// TwinCAT 3 PLC project EpicsComModule
// ProgramVersion: 3.1.4022.2
// libraries:
//   Tc2_EtherCAT, * (Beckhoff Automation GmbH)
//   Tc2_Standard, * (Beckhoff Automation GmbH)
//   Tc2_System, * (Beckhoff Automation GmbH)
//   Tc2_TcpIp, * (Beckhoff Automation GmbH)
//   Tc2_Utilities, * (Beckhoff Automation GmbH)
//   Tc3_Interfaces, * (Beckhoff Automation GmbH)
//   Tc3_Module, * (Beckhoff Automation GmbH)
// project tree:
//   Data types/ DUT_AxisStatus_v0_01.TcDUT, E_ConnectionSteps.TcDUT, E_ServerSteps.TcDUT, DUT_ComSettings.TcDUT
//   Global Variables/ Global_Variables.TcGVL
//   / PlcTaskCom.TcTTO
//   POUs/DUT_Support/ FB_Read_DUT_AxisStatus_v0_01.TcPOU
//   POUs/ FB_ServerApplication.TcPOU, FB_ServerConnection.TcPOU, FB_Server.TcPOU, FB_StreamBufferToADSBuffer.TcPOU, FB_ValidCommand.TcPOU, FB_ADSBufferToStreamBuffer.TcPOU, MAIN.TcPOU, README.TcPOU
//   POUs/Helper POUs/ CheckBounds.TcPOU, FB_FindChar.TcPOU, FB_FrameFifo.TcPOU, FB_LogFifo.TcPOU, F_RemoveBytesFromBuffer.TcPOU
//   POUs/Static Command support/ FB_GetStaticADR.TcPOU, FB_ParseStaticCommand.TcPOU, FB_ParseStringToSymInfo.TcPOU, FB_SetStaticADSPort.TcPOU, FB_SetStaticADR.TcPOU, FB_ParseCommandOption.TcPOU

CONFIGURATION EpicsComModule
    RESOURCE PLC ON TwinCAT3
        TASK PlcTaskCom(INTERVAL := T#1ms, PRIORITY := 26);
        PROGRAM MAIN WITH PlcTaskCom : MAIN;
    END_RESOURCE
END_CONFIGURATION

// ---- Data types/DUT_AxisStatus_v0_01.TcDUT
TYPE DUT_AxisStatus_v0_01:
STRUCT
    bEnable: BOOL;
    bReset: BOOL;
    bExecute: BOOL;
    nCommand: UINT;
    nCmdData: UINT;
    fVelocity: LREAL;
    fPosition: LREAL;
    fAcceleration: LREAL;
    fDeceleration: LREAL;
    bJogFwd: BOOL;
    bJogBwd: BOOL;
    bLimitFwd: BOOL;
    bLimitBwd: BOOL;
    fOverride: LREAL:=100;
    bHomeSensor: BOOL;
    bEnabled: BOOL;
    bError: BOOL;
    nErrorId: UDINT;
    fActVelocity: LREAL;
    fActPosition: LREAL;
    fActDiff: LREAL;
    bHomed:BOOL;
    bBusy:BOOL;
END_STRUCT
END_TYPE

// ---- Data types/E_ConnectionSteps.TcDUT
TYPE E_ConnectionSteps :
(
    eCONNECTION_STATE_IDLE,
    eCONNECTION_STATE_CONNECT_START,
    eCONNECTION_STATE_CONNECT_WAIT,
    eCONNECTION_STATE_DATAEXCHANGE,
    eCONNECTION_STATE_CLOSE_START,
    eCONNECTION_STATE_CLOSE_WAIT,
    eCONNECTION_STATE_ERROR
);
END_TYPE

// ---- Data types/E_ServerSteps.TcDUT
TYPE E_ServerSteps :
(
    eSERVER_STATE_IDLE,
    eSERVER_STATE_LISTENER_OPEN_START,
    eSERVER_STATE_LISTENER_OPEN_WAIT,
    eSERVER_STATE_REMOTE_CLIENTS_COMM,
    eSERVER_STATE_REMOTE_CLIENTS_CLOSE,
    eSERVER_STATE_LISTENER_CLOSE_START,
    eSERVER_STATE_LISTENER_CLOSE_WAIT,
    eSERVER_STATE_ERROR
);
END_TYPE

// ---- Data types/DUT_ComSettings.TcDUT
TYPE DUT_ComSettings :
STRUCT
    nConnectionIndex:UDINT:=0;
    nADSPort:INT:=851;
    bReturnData:BOOL:=FALSE;
    bReturnVarName:BOOL:=FALSE;
END_STRUCT
END_TYPE

// ---- Global Variables/Global_Variables.TcGVL
VAR_GLOBAL CONSTANT
    MAX_CLIENT_CONNECTIONS                  : UDINT(1..20) := 5;
    PLCPRJ_BUFFER_SIZE                      : UDINT := 20000;(* Max. internal fifo/receiver buffer size *)
    PLCPRJ_RECEIVE_POLLING_TIME             : TIME := T#1MS; //Changed from example where it was 1000ms. => epics timeout all the time!
    PLCPRJ_RECEIVE_TIMEOUT                  : TIME := T#0S;

    (* Some project specific error codes *)
    PLCPRJ_ERROR_RECEIVE_TIMEOUT            : UDINT := 16#8101;(* Receive timeout *)
    PLCPRJ_ERROR_SENDFIFO_OVERFLOW          : UDINT := 16#8102;(* Send fifo overflow *)
    PLCPRJ_ERROR_RECFIFO_OVERFLOW           : UDINT := 16#8103;(* Receive fifo overflow *)

    //EPICS related constants
    EPICS_MAX_FRAME_SIZE                    : INT :=1400; //Max size of variable string (for communication with epics) Arrays can be divided in several frames/stings (atleast for reading operation)
    EPICS_ARRAY_DELIMITER                   : STRING :=',';
    EPICS_COMMAND_DELIMITER                 : STRING := ';';
    EPICS_READ_CMD                          : STRING:= '?';
    EPICS_WRITE_CMD                         : STRING:= '=';
    EPICS_ACK_STRING                        : STRING:='OK';
    EPICS_ASCII_DOT                         : BYTE:=46;
    EPICS_ASCII_LN                          : BYTE:=10;
    EPICS_ASCII_CR                          : BYTE:=13;
    EPICS_ASCII_COMMA                       : BYTE:=44;     // Must be same as EPICS_ARRAY_DELIMITER. This variable should be autoamtically genrated instead. Maybe in next version?!
    EPICS_ASCII_ZERO                        : BYTE:=48;
    EPICS_ASCII_ONE                         : BYTE:=49;
    EPICS_ASCII_EQUAL                       : BYTE:=61;     // Must be same as EPICS_WRITE_CMD. This variable should be autoamtically genrated instead. Maybe in next version?!
    EPICS_ASCII_QUESTIONMARK                : BYTE:=63;     // Must be same as EPICS_READ_CMD. This variable should be autoamtically genrated instead. Maybe in next version?!
    EPICS_ASCII_COMMAND_DELIMITER           : BYTE:=59;     // Must be same as EPICS_COMMAND_DELIMITER. This variable should be autoamtically genrated instead. Maybe in next version?!
    EPICS_COM_TIMEOUT                       : TIME:=T#1S;   // Not used yet
    EPICS_MAX_STACKED_STATIC_COMMANDS       : INT:=5;       // Maximum options to command

    //Command Options
    EPICS_COMMAND_OPTION_DELIMITER          : STRING := '/';        //Used for static commands that should not excute symboliclly
    EPICS_COMMAND_OPTION_ADSPORT            : STRING := 'ADSPORT';  //USED to set ADS port from command. Applicable only for this command

    //Static Commands
    EPICS_STATIC_COMMAND_TRIGGER            : STRING := '.';        //Setting for return of data for write commands (data instead of "OK;"). Applicable only for this command
    EPICS_STATIC_COMMAND_THIS               : STRING := 'THIS.';    //Setting for return of data for write commands (data instead of "OK;"). Applicable only for this command
    EPICS_STATIC_COMMAND_THIS_PATH          : STRING := 'Main.fbServer.aApplications';  //Setting for return of data for write commands (data instead of "OK;"). Applicable only for this command
    EPICS_STATIC_COMMAND_ADR                : STRING := 'ADR.';     //Setting for return of data for write commands (data instead of "OK;"). Applicable only for this command

END_VAR

VAR_GLOBAL
        EPICS_SAMPLE_TIME                   : INT:=1;       // The EPICS COM module will be executed every EPICS_SAMPLE_TIME cycle
        EPICS_FORMAT_ASCII                  : BOOL:=TRUE;   // Not used yet. Binary transfer of data is not currently supported.
END_VAR

// ---- POUs/MAIN.TcPOU
///#########################################################
///Main POU for TCP/IP based EPICS-interface. The TCP/IP server related code is based on Beckhoff sample code. Changes and additions have been made to this code for the general purpose EPICS interface.
///
/// Library:
///
///
/// Global Variables:
/// - EPICS_MAX_FRAME_SIZE
/// - EPICS_ARRAY_DELIMITER
/// - EPICS_COMMAND_DELIMITER
/// - PLCPRJ_BUFFER_SIZE
///
/// Data types:
///
/// External functions:
///     - TC2_Standard lib
///     - Tc2_Utilities lib
///     - Tc2_System lib
///
///
///###########################################################

PROGRAM MAIN
VAR
    sVersion: STRING:='0.9.1';
END_VAR
VAR
    sSrvNetID   : T_AmsNetID    := '';(* TwinCAT TCP/IP server network address *)
    bEnable     : BOOL := TRUE;(* TRUE => Enable server data exchange, FALSE => Disable *)
    bLog        : BOOL := FALSE;(* TRUE => Enable message/error log, FALSE => Disable *)

    fbServer    : FB_Server := (    sLocalHost :=  '0.0.0.0' (*Own (server) IP address!  '192.168.40.106'*),
                                    nLocalPort := 5000,(* Own (server) port number! *)
                                    sPrefix := 'SERVER::' );

    fbCloseAll  : FB_SocketCloseAll;
    bInitialize : BOOL := TRUE;

    //Included utilities in EpicsComModule
    fbNTShutdown: NT_Shutdown;
    fbNTAbortShutdown:NT_AbortShutdown;
    iCounter:INT:=0;
    bErrorWritten:BOOL:=FALSE;
    sErrorMessage:STRING(255);
END_VAR

//Delay execution
IF EPICS_SAMPLE_TIME>100 THEN
    EPICS_SAMPLE_TIME:=100;
ELSIF  EPICS_SAMPLE_TIME<1 THEN
    EPICS_SAMPLE_TIME:=1;
END_IF

iCounter:=iCounter+1;
IF iCounter>=EPICS_SAMPLE_TIME THEN  //Possability to change communcation execution speed from EPICS (via the global variable EPICS_SAMPLE_TIME)
    iCounter:=0;
    (* On PLC reset or program download close all created/opened sockets/connections *)
    fbCloseAll( sSrvNetID := sSrvNetID, bExecute:= bInitialize );
    IF fbCloseAll.bError AND NOT bErrorWritten THEN
        sErrorMessage:=UDINT_TO_STRING(fbCloseAll.nErrId);
        ADSLOGSTR( ADSLOG_MSGTYPE_ERROR, 'EPICSComModule: fbCloseAll failed with errorId %s.', sErrorMessage);
        bErrorWritten:=TRUE;
    END_IF
    IF fbCloseAll.bBusy OR fbCloseAll.bError THEN
        RETURN;
    END_IF
    bErrorWritten:=FALSE;
    bInitialize := FALSE;
    fbServer( sSrvNetID := sSrvNetID, bEnable := bEnable, bLog := bLog );
END_IF

//Execution of utilities Action
Utilities();

ACTION Utilities:
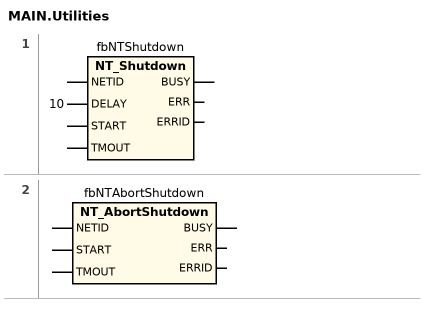
// NETWORK 1
//   fbNTShutdown: Included utilities in EpicsComModule
fbNTShutdown(DELAY := 10); // NT_Shutdown

// NETWORK 2
fbNTAbortShutdown(); // NT_AbortShutdown
END_ACTION

END_PROGRAM

// ---- POUs/FB_Server.TcPOU
///#########################################################
///FB that handles TCP/IP server and the client connections. The code is based on Beckhoff sample code. However changes and additions have been made to this code for the general purpose EPICS interface.
///
///
/// Library:
///
/// Global Variables:
/// - EPICS_MAX_FRAME_SIZE
/// - EPICS_ARRAY_DELIMITER
/// - EPICS_COMMAND_DELIMITER
/// - PLCPRJ_BUFFER_SIZE
///
/// Data types:
///
/// External functions:
///     - TC2_Standard lib
///     - Tc2_Utilities lib
///     - Tc2_System lib
///
///###########################################################

FUNCTION_BLOCK FB_Server
VAR
    sVersion: STRING:='0.9.1';
END_VAR
VAR_INPUT
    sSrvNetID       : T_AmsNetID    := '';(* TwinCAT TCP/IP server network address *)
    sLocalHost      : T_IPv4Addr    := '127.0.0.1';(* Own IP address! *)
    nLocalPort      : UDINT         := 0;(* Server port number *)
    bEnable         : BOOL          := FALSE;(* TRUE => enable server data exchange, FALSE => disable *)
    tReconnect      : TIME          := T#3S;(* Reopen new listener socket after this time *)
    bLog            : BOOL          := FALSE;(* TRUE => Enable log message output, FALSE => Disable *)
    sPrefix         : STRING        := 'SERVER::';(* Log message description string (allows the identification of log message source) *)
END_VAR
VAR_OUTPUT
    bListening      : BOOL          := FALSE;(* Listener socket state *)
    nAccepted       : UDINT         := 0;(* Max. number of accepted client connections *)
END_VAR
VAR
    aApplications   : ARRAY[1..MAX_CLIENT_CONNECTIONS] OF FB_ServerApplication;(* Server application control function blocks *)
    aConnections    : ARRAY[1..MAX_CLIENT_CONNECTIONS] OF FB_ServerConnection :=
                                                    [   (sPrefix := 'SERVER1::'),
                                                        (sPrefix := 'SERVER2::'),
                                                        (sPrefix := 'SERVER3::'),
                                                        (sPrefix := 'SERVER4::'),
                                                        (sPrefix := 'SERVER5::') ];(* Server connection/data exchange control function blocks *)
    aTx             : ARRAY[1..MAX_CLIENT_CONNECTIONS] OF FB_FrameFifo;(* TX fifo *)
    aRx             : ARRAY[1..MAX_CLIENT_CONNECTIONS] OF FB_FrameFifo;(* RX fifo *)
    aLog            : ARRAY[1..MAX_CLIENT_CONNECTIONS] OF FB_LogFifo;(* Listener log message fifo *)
    fbListen        : FB_SocketListen;
    fbClose         : FB_SocketClose;
    fbLog           : FB_LogFifo;
    fbListenTimer   : TON;
    bReset          : BOOL := FALSE;
    eStep           : E_ServerSteps;
    i               : UDINT;
END_VAR



CASE eStep OF
    eSERVER_STATE_IDLE:
        IF bEnable XOR bListening THEN
            IF bEnable THEN
                fbListenTimer( IN := TRUE );
                IF fbListenTimer.Q THEN
                    fbListenTimer( IN := FALSE, PT := tReconnect );

                    fbLog.Clear( sPrefix := sPrefix, bLog := bLog );(* Clear listener log fifo *)
                    bReset := FALSE;

                    eStep := eSERVER_STATE_LISTENER_OPEN_START;
                END_IF
            ELSE
                eStep := eSERVER_STATE_REMOTE_CLIENTS_CLOSE;
            END_IF
        ELSIF bListening THEN
            eStep := eSERVER_STATE_REMOTE_CLIENTS_COMM;
        ELSE
            fbListenTimer( IN := FALSE, PT := T#0S );
            bReset := FALSE;
        END_IF

    eSERVER_STATE_LISTENER_OPEN_START:
        fbListen(  bExecute := FALSE  );
        fbListen(   sSrvNetID := sSrvNetID,
                    sLocalHost := sLocalHost,
                    nLocalPort := nLocalPort,
                    bExecute := TRUE );
        eStep := eSERVER_STATE_LISTENER_OPEN_WAIT;

    eSERVER_STATE_LISTENER_OPEN_WAIT:
        fbListen( bExecute := FALSE );
        IF NOT fbListen.bBusy THEN
            IF NOT fbListen.bError THEN
                bListening  := TRUE;
                fbLog.Message( sMessage := 'Listener socket opened!', hSocket := fbListen.hListener );
                eStep := eSERVER_STATE_IDLE;
            ELSE
                fbLog.Error( sMessage := 'FB_SocketListen()', nErrId := fbListen.nErrId );
                eStep := eSERVER_STATE_ERROR;
            END_IF
        END_IF

    eSERVER_STATE_REMOTE_CLIENTS_COMM:
        eStep := eSERVER_STATE_IDLE;
        nAccepted := 0;

        FOR i:= 1 TO MAX_CLIENT_CONNECTIONS DO
            aApplications[i].nConnectionIndex:=i;
            aConnections[i]( fbTx := aTx[i], fbRx := aRx[i], fbLog := aLog[i],
                            hListener := fbListen.hListener, bReset := bReset,
                            sSrvNetID := sSrvNetID, bEnable := bEnable, bLog := bLog );
            IF bReset THEN
                bReset := FALSE;
                eStep := eSERVER_STATE_REMOTE_CLIENTS_CLOSE;
                EXIT;
            END_IF

            IF aConnections[i].bAccepted THEN
                aApplications[i]( fbTx := aTx[i], fbRx := aRx[i], fbLog := aLog[i]);
                nAccepted := nAccepted + 1;(* Count the number of connected remote clients *)
                aApplications[i].bReset:=FALSE;
            ELSE
                    aApplications[i].bReset:=TRUE;
                    aApplications[i]( fbTx := aTx[i], fbRx := aRx[i], fbLog := aLog[i]);
            END_IF


        END_FOR

    eSERVER_STATE_REMOTE_CLIENTS_CLOSE:
        nAccepted := 0;
        FOR i:= 1 TO MAX_CLIENT_CONNECTIONS DO
            (* Close all remote client (accepted) sockets *)
            aConnections[i]( fbTx := aTx[i], fbRx := aRx[i], fbLog := aLog[i],
                            hListener := fbListen.hListener, bReset := bReset,
                            sSrvNetID := sSrvNetID, bEnable := FALSE, bLog := bLog );
            IF aConnections[i].bAccepted THEN
                nAccepted := nAccepted + 1;(* Count the number of connected remote clients *)
            END_IF
        END_FOR

        (* Check if all remote client sockets are closed *)
        IF nAccepted = 0 THEN
            eStep := eSERVER_STATE_LISTENER_CLOSE_START; (* Close listener socket too *)
        END_IF

    eSERVER_STATE_LISTENER_CLOSE_START:
        fbLog.Message( sMessage := 'Closing listener socket!', hSocket := fbListen.hListener );
        fbClose( bExecute := FALSE );
        fbClose( sSrvNetID := sSrvNetID, hSocket := fbListen.hListener, bExecute:= TRUE );
        eStep := eSERVER_STATE_LISTENER_CLOSE_WAIT;

    eSERVER_STATE_LISTENER_CLOSE_WAIT:
        fbClose( bExecute := FALSE );
        IF NOT fbClose.bBusy THEN
            bListening := FALSE;
            nAccepted := 0;
            IF NOT fbClose.bError THEN
                eStep := eSERVER_STATE_IDLE;
            ELSE
                fbLog.Error( sMessage := 'FB_SocketClose(listener)', nErrId := fbListen.nErrID );
                eStep := eSERVER_STATE_ERROR;
            END_IF
        END_IF

    eSERVER_STATE_ERROR:
        IF bListening THEN
            eStep := eSERVER_STATE_REMOTE_CLIENTS_CLOSE;
        ELSE
            eStep := eSERVER_STATE_IDLE;
        END_IF

END_CASE

END_FUNCTION_BLOCK

// ---- POUs/FB_ServerApplication.TcPOU
///#########################################################
///FB that handles one EPICS connection of TCP/IP.
/// The main functionallity of this function block is to parse commands from EPICS or other serial device.
///
/// Library:
///
///
/// Global Variables:
/// - EPICS_MAX_FRAME_SIZE
/// - EPICS_ARRAY_DELIMITER
/// - EPICS_COMMAND_DELIMITER
/// - PLCPRJ_BUFFER_SIZE
///
/// Data types:
///
/// External functions:
///     - TC2_Standard lib
///     - Tc2_Utilities lib
///     - Tc2_System lib
///
///###########################################################
FUNCTION_BLOCK FB_ServerApplication
VAR
    sVersion: STRING:='0.9.1';
    sFeatures: STRING:='stv1';
END_VAR
VAR_IN_OUT
    fbTx        : FB_FrameFifo;(* TX fifo *)
    fbRx        : FB_FrameFifo;(* RX fifo *)
    fbLog       : FB_LogFifo;(* Log message fifo *)
END_VAR

VAR_INPUT
    nConnectionIndex:UDINT:=0;
    bReset: BOOL;
END_VAR

VAR
    //Settings
    nADSPort                            : UINT:=851;
    nState                              :INT:=0;

    bExecuteWriteBufferToEPICS:BOOL:=FALSE;
    bInStaticSection:BOOL:=FALSE;
    bReadCmd: BOOL:=FALSE;
    bWriteCmd: BOOL:=FALSE;
    bStaticGetADRCommand    :   BOOL:=FALSE;
    bStaticTHISCommand      :   BOOL:=FALSE;

    //FB:s
    fbAdsReadValue: Tc2_System.ADSREAD;
    fbAdsWriteValue: Tc2_System.ADSWRITE;
    fbParseADSBufferToStream:FB_ADSBufferToStreamBuffer;
    fbParseStreamBufferToADS:FB_StreamBufferToADSBuffer;
    fbStateTimoutTimer:TON;
    fbSymInfoByName:Tc2_Utilities.PLC_ReadSymInfoByName;
    fbValidCommand:FB_ValidCommand;
    fbParseCommandOption:FB_ParseCommandOption;
    fbParseStringToSymInfo: FB_ParseStringToSymInfo;
    stSettings: DUT_ComSettings;
    fbFincChar: FB_FindChar;
    //buffers
    byteADSBuffer       : ARRAY[0..PLCPRJ_BUFFER_SIZE] OF BYTE;
    byteCommandBuffer   : ARRAY[0..PLCPRJ_BUFFER_SIZE] OF BYTE; (* Byte buffer*)
    byteFrameBuffer     : ARRAY[0..EPICS_MAX_FRAME_SIZE] OF BYTE;

    //Strings
    sTemp: STRING;
    sAckString: STRING;
    psCommandBufferString: POINTER TO STRING; //string to point into byte buffer
    sVariableName: STRING;

    //Ints
    nBytesInCommandBuffer:DINT;
    nADSBytesToRead: DINT;
    nIndexEndOfCommand: DINT;
    nIndex1:INT:=0;
    nLength: INT;

    //Error handling
    sComBufferAtError: STRING;
    sError: STRING(255);
    sSubErrorString:STRING(255);
    bErrorMessageSent: BOOL:=FALSE;
    bErrorOld: BOOL;
    nErrorCounter: INT;
    stSymInfo:SYMINFOSTRUCT;
    nStatricCommandCounter: INT;
    sGetStaticADR:STRING(255):='';
    iEmptyCounter: INT;
    nFrameBufferIndex: INT;
    nCleanBytes: DINT;
    sVariableName_THIS: STRING(INT#255);
    sVarName: STRING(INT#255);
    nLengthSubString: INT;
END_VAR

VAR_OUTPUT
    nErrorId: UDINT;
    bError: BOOL;
END_VAR



//Typical command string: "ADSPORT=851/Main.M1.fPosition=100;ADSPORT=852/Main.iCounter?;linefeed"

psCommandBufferString :=ADR(byteCommandBuffer[0]); //Used for debugging to see byte buffer as string
stSettings.nConnectionIndex:=nConnectionIndex;

//State 1: Get new info from recieve buffer. Wait for complete command = ";"
IF nState=0 THEN //Only get new data from buffer if free mem
    fbRx.RemoveHead(bGet := ADR(byteCommandBuffer[nBytesInCommandBuffer]), nReadBufferSize:=SIZEOF(byteCommandBuffer)-nBytesInCommandBuffer);(* Fetch string from rx fifo *)
    IF fbRx.bOk THEN(* Success *)
        nBytesInCommandBuffer:=nBytesInCommandBuffer+DINT_TO_INT(fbRx.nReadCount); //Seems buffer always returns one byte less thann count?
        //fbLog.Error( sMessage := concat(str1:='State 1a: ', str2:=PSTRING_TO_STRING(psCommandBufferString)), nErrID := nBytesInCommandBuffer );
    END_IF
END_IF

IF  nBytesInCommandBuffer>0 AND NOT (nState=1) THEN
    fbValidCommand(nBytesInCommandBuffer:=nBytesInCommandBuffer,pbCommandBuffer:=ADR(byteCommandBuffer));
    //fbLog.Error( sMessage := concat(str1:='State 1b: ', str2:=PSTRING_TO_STRING(psCommandBufferString)), nErrID := nBytesInCommandBuffer );
    IF  fbValidCommand.bValid THEN
        nIndexEndOfCommand:=fbValidCommand.nIndexEndOfCommand;
        nState:=1;
    END_IF
END_IF

//State 2: Check for Command Options
IF (nState=1) THEN
    //Reset defaults
    nADSPort:=stSettings.nADSPort;
    nStatricCommandCounter:=0;
    bInStaticSection:=TRUE;
    REPEAT
        nStatricCommandCounter:=nStatricCommandCounter+1;
        nIndex1:=find(STR1:=PSTRING_TO_STRING(psCommandBufferString),STR2:=EPICS_COMMAND_OPTION_DELIMITER);

        IF nIndex1>0 AND nIndex1<=nIndexEndOfCommand THEN
            fbParseCommandOption(nCommandEndIndex:=nIndex1,byteCommandBuffer:=byteCommandBuffer,nBytesInCommandBuffer:=nBytesInCommandBuffer,nIndexEndOfCommand:=nIndexEndOfCommand);
            IF NOT fbParseCommandOption.bError THEN
                IF len(fbParseCommandOption.sStaticCommand)>0 THEN
                    //*****EPICS_COMMAND_OPTION_ADSPORT
                    IF find(STR1:=fbParseCommandOption.sStaticCommand,STR2:=EPICS_COMMAND_OPTION_ADSPORT)>0 THEN
                        IF fbParseCommandOption.bWriteCommand THEN
                            nADSPort:=STRING_TO_UINT(fbParseCommandOption.sStaticValue);
                        END_IF
                    END_IF
                END_IF
            ELSE
                bError:=fbParseCommandOption.bError;
                sSubErrorString:=fbParseCommandOption.sSubErrorString;
                nErrorId:=fbParseCommandOption.nErrorId;
            END_IF
        ELSE
            bInStaticSection:=FALSE;
        END_IF
    UNTIL nBytesInCommandBuffer<1 OR (NOT bInStaticSection) OR bError OR nStatricCommandCounter>EPICS_MAX_STACKED_STATIC_COMMANDS OR nIndex1=0
    END_REPEAT
    IF NOT bError THEN
        nState:=2;
    END_IF
    //fbLog.Error( sMessage := concat(str1:='State 2: ', str2:=PSTRING_TO_STRING(psCommandBufferString)), nErrID := nBytesInCommandBuffer );
END_IF

//State 3: Check if Static Commands
IF (nState=2) THEN
    bStaticTHISCommand:=FALSE;
    bStaticGetADRCommand:=FALSE;
    nIndex1:=find(STR1:=PSTRING_TO_STRING(psCommandBufferString),STR2:=EPICS_STATIC_COMMAND_TRIGGER);
    IF (nIndex1=1) THEN
         //Command EPICS_STATIC_COMMAND_THIS = "#THIS."
        nIndex1:=find(STR1:=PSTRING_TO_STRING(psCommandBufferString),STR2:=EPICS_STATIC_COMMAND_THIS);
        IF (nIndex1=2) THEN   //Command should be = "#THIS."
            //=
            nIndex1:=find(STR1:=PSTRING_TO_STRING(psCommandBufferString),STR2:=EPICS_WRITE_CMD);        //=
            IF nIndex1<1 OR nIndex1 > nIndexEndOfCommand THEN
                nIndex1:=find(STR1:=PSTRING_TO_STRING(psCommandBufferString),STR2:=EPICS_READ_CMD); //?
            END_IF
            //Remove static commands and build variable name to this fb. (this.stSettings.nPort=>Main.fbServer.aApplications[nConnectionIndex].stSettings.nPort)
            stemp:=left(str:=PSTRING_TO_STRING(psCommandBufferString),SIZE:=nIndex1-1);
            stemp:=right(str:=sTemp,size:=len(sTemp)-(len(EPICS_STATIC_COMMAND_TRIGGER)+len(EPICS_STATIC_COMMAND_THIS)));
            sVariableName_THIS:=concat(STR1:=EPICS_STATIC_COMMAND_THIS_PATH,STR2:='[');
            sVariableName_THIS:=concat(STR1:=sVariableName_THIS,STR2:=UDINT_TO_STRING(nConnectionIndex));
            sVariableName_THIS:=concat(STR1:=sVariableName_THIS,STR2:='].');
            sVariableName_THIS:=concat(STR1:=sVariableName_THIS,STR2:=sTemp);
            bStaticTHISCommand:=TRUE;
            //Don't clean up this command. Will be done in subsequent steps
        ELSE
             //Command EPICS_STATIC_COMMAND_THIS = "#ADR."
            nIndex1:=find(STR1:=PSTRING_TO_STRING(psCommandBufferString),STR2:=EPICS_STATIC_COMMAND_ADR);
            IF (nIndex1=2) THEN   //Command should be = "#ADR."
                //= write. Expect a command like:  "#ADR.1,1,1,1=200;"
                nIndex1:=find(STR1:=PSTRING_TO_STRING(psCommandBufferString),STR2:=EPICS_WRITE_CMD);        //=
                IF (nIndex1>0) AND ((nIndex1-1) < nIndexEndOfCommand) THEN
                    bWriteCmd:=TRUE;
                ELSE
                    //? read. Expect a command like:  "#ADR.1,1,1,1?;" => ask for value, or "#ADR.Main.M1.bEnable?;"=> ask for adress
                    nIndex1:=find(STR1:=PSTRING_TO_STRING(psCommandBufferString),STR2:=EPICS_READ_CMD);     //?
                    IF ((nIndex1>0) AND (nIndex1-1) < nIndexEndOfCommand) THEN
                        bReadCmd:=TRUE;
                    END_IF
                END_IF
                IF bReadCmd OR bWriteCmd THEN
                    sVariableName:=left(str:=PSTRING_TO_STRING(psCommandBufferString),SIZE:=nIndex1-1);
                    sVariableName:=right(str:=sVariableName,size:=len(sVariableName)-(len(EPICS_STATIC_COMMAND_TRIGGER)+len(EPICS_STATIC_COMMAND_ADR)));
                    //Check if symbol or abs adress
                    nLengthSubString:=(len(EPICS_STATIC_COMMAND_ADR)+len(EPICS_STATIC_COMMAND_TRIGGER));
                    fbFincChar(pbBuffer:=ADR(byteCommandBuffer[0]),nLength:=nIndex1,cFind:=EPICS_ASCII_DOT,nStartIndex:=nLengthSubString+2);
                    IF ((fbFincChar.nIndex>nLengthSubString) AND (fbFincChar.nIndex-1) <nIndexEndOfCommand) THEN
                        bStaticGetADRCommand:=TRUE;
                        nState:=4;  // return abs.-adress for symbolic adress
                    ELSE
                        fbParseStringToSymInfo(sAdress:=sVariableName);
                        IF NOT fbParseStringToSymInfo.bError THEN
                            stSymInfo:=fbParseStringToSymInfo.stSymInfo;
                            nState:=5;
                        ELSE
                            bError:=fbParseStringToSymInfo.bError;
                            nErrorId:=fbParseStringToSymInfo.nErrorId;
                            sSubErrorString:=fbParseStringToSymInfo.sSubErrorString;
                        END_IF
                    END_IF
                    IF NOT F_RemoveBytesFromBuffer(nIndex1,byteCommandBuffer:=byteCommandBuffer,nBytesInCommandBuffer:=nBytesInCommandBuffer,nIndexEndOfCommand:=nIndexEndOfCommand) THEN
                            bError:=TRUE;
                            nErrorId:=301;
                            sSubErrorString:='State 3: Failed to clear buffer (read).';
                    END_IF
                END_IF
            END_IF
        END_IF
    END_IF
    IF (NOT bError) AND (nState<3) THEN
        nState:=3;
    END_IF
    //fbLog.Error( sMessage := concat(str1:='State 3: ', str2:=PSTRING_TO_STRING(psCommandBufferString)), nErrID := nBytesInCommandBuffer );
END_IF

//State 4: Find symbolic variable name in cmd
IF (nState=3) THEN
    //check if read cmd
    bReadCmd:=FALSE;
    bWriteCmd:=FALSE;
    nIndex1:=find(STR1:=PSTRING_TO_STRING(psCommandBufferString),STR2:=EPICS_READ_CMD);
    IF nIndex1>0 AND nIndex1<= nIndexEndOfCommand THEN
        sVariableName:=left(STR:=PSTRING_TO_STRING(psCommandBufferString), SIZE:=nIndex1-1);
        //Clear buffer
        IF F_RemoveBytesFromBuffer(nIndex1,byteCommandBuffer:=byteCommandBuffer,nBytesInCommandBuffer:=nBytesInCommandBuffer,nIndexEndOfCommand:=nIndexEndOfCommand) THEN
            bReadCmd:=TRUE;
        ELSE
            bError:=TRUE;
            nErrorId:=402;
            sSubErrorString:='State 4: Failed to clear buffer (read).';
        END_IF
    ELSE
        nIndex1:=find(STR1:=PSTRING_TO_STRING(psCommandBufferString),STR2:=EPICS_WRITE_CMD);
        IF nIndex1>0 AND nIndex1<=nIndexEndOfCommand THEN
            sVariableName:=left(STR:=PSTRING_TO_STRING(psCommandBufferString), SIZE:=nIndex1-1);
            IF F_RemoveBytesFromBuffer(nIndex1,byteCommandBuffer:=byteCommandBuffer,nBytesInCommandBuffer:=nBytesInCommandBuffer,nIndexEndOfCommand:=nIndexEndOfCommand) THEN
                bWriteCmd:=TRUE;
            ELSE
                bError:=TRUE;
                nErrorId:=403;
                sSubErrorString:='State 4: Failed to clear buffer (write).';
            END_IF
        END_IF
    END_IF
    IF bWriteCmd OR bReadCmd THEN
        nState:=4;
    END_IF
    IF NOT bError THEN
        IF NOT (nState=4) THEN
            bError:=TRUE;
            nErrorId:=401;
            sSubErrorString:='State 4: No read or write command identified.';
        END_IF
    END_IF;
    fbSymInfoByName(START:=FALSE);
    //fbLog.Error( sMessage := concat(str1:='State 4: ', str2:=PSTRING_TO_STRING(psCommandBufferString)), nErrID := nBytesInCommandBuffer );
END_IF


//State 5: Get symbolic information over ADS
IF (nState=4) THEN
    //If static command "THIS" then use other variable name
    IF bStaticTHISCommand THEN
        sVarName:=sVariableName_THIS;
    ELSE
        sVarName:=sVariableName;
    END_IF
    fbSymInfoByName(
            PORT:= nADSPort,
            SYMNAME:= sVarName,
            START:= TRUE,
            TMOUT:=T#100MS);

        (*Wait until it's done or if an error occurs*)
        IF NOT fbSymInfoByName.ERR THEN
            IF NOT fbSymInfoByName.BUSY THEN
                nState:=5;
                stSymInfo:=fbSymInfoByName.SYMINFO;
                fbAdsReadValue(read:=FALSE);
                IF bStaticGetADRCommand THEN // jump over next state and prepare information to be sent
                    sGetStaticADR:='';
                    sGetStaticADR:=CONCAT(str1:=sGetStaticADR,str2:='16#');
                    sGetStaticADR:=CONCAT(str1:=sGetStaticADR,str2:=DWORD_TO_HEXSTR(stSymInfo.idxGroup,1,FALSE));
                    sGetStaticADR:=CONCAT(str1:=sGetStaticADR,str2:=EPICS_ARRAY_DELIMITER);
                    sGetStaticADR:=CONCAT(str1:=sGetStaticADR,str2:='16#');
                    sGetStaticADR:=CONCAT(str1:=sGetStaticADR,str2:=DWORD_TO_HEXSTR(stSymInfo.idxOffset,1,FALSE));
                    sGetStaticADR:=CONCAT(str1:=sGetStaticADR,str2:=EPICS_ARRAY_DELIMITER);
                    sGetStaticADR:=CONCAT(str1:=sGetStaticADR,str2:=DINT_TO_STRING(stSymInfo.byteSize));
                    sGetStaticADR:=CONCAT(str1:=sGetStaticADR,str2:=EPICS_ARRAY_DELIMITER);
                    sGetStaticADR:=CONCAT(str1:=sGetStaticADR,str2:=DINT_TO_STRING(stSymInfo.adsDataType));
                    nFrameBufferIndex:=len(sGetStaticADR);
                    stSymInfo.byteSize:=len(str:=sGetStaticADR);        //Fake size
                    memcpy(destAddr:=ADR(byteADSBuffer[0]),srcAddr:=ADR(sGetStaticADR),n:=stSymInfo.byteSize);  //Copy to output buffer
                    stSymInfo.adsDataType :=ADST_STRING;                //Fake string
                    bReadCmd:=TRUE;
                    nState:=8;                                          //Jump to state 9
                    bExecuteWriteBufferToEPICS:=TRUE;                   //Execute write directly size all info is prepared
                END_IF
            END_IF
        ELSE
            bError:=TRUE;
            nErrorId:=fbSymInfoByName.ERRID;
            sSubErrorString:=concat(str1:='State 5: Failed to get symbolic information for variable:',STR2:=sVariableName);
        END_IF;
        //fbLog.Error( sMessage := concat(str1:='State 5: ', str2:=PSTRING_TO_STRING(psCommandBufferString)), nErrID := nBytesInCommandBuffer );
END_IF

//State 6: Convert stream buffer to ADS buffer (WRITE)
IF (nState=5) AND bWriteCmd THEN
    //fbLog.Error( sMessage := concat(str1:='State 6: ', str2:=PSTRING_TO_STRING(psCommandBufferString)), nErrID := nBytesInCommandBuffer );
    fbParseStreamBufferToADS(bExecute:=TRUE,symbolInfo:=stSymInfo,nBufferToParseLength:=nIndexEndOfCommand,fbLog:=fbLog,byteASCIIBufferToParse:=byteCommandBuffer,byteBinayBufferOutput:=byteADSBuffer);
    IF NOT fbParseStreamBufferToADS.bError  THEN
        IF NOT fbParseStreamBufferToADS.bBusy THEN
            nCleanBytes:=fbParseStreamBufferToADS.nASCIIBytesParsed;
            IF nCleanBytes>0 AND nCleanBytes+fbParseStreamBufferToADS.nASCIIBytesParsed < PLCPRJ_BUFFER_SIZE-255 THEN
                F_RemoveBytesFromBuffer(nCleanBytes,byteCommandBuffer:=byteCommandBuffer,nBytesInCommandBuffer:=nBytesInCommandBuffer,nIndexEndOfCommand:=nIndexEndOfCommand);
                fbAdsWriteValue(WRITE:=FALSE);
                nState:=6;
                fbParseStreamBufferToADS(bExecute:=FALSE,symbolInfo:=stSymInfo,nBufferToParseLength:=nIndexEndOfCommand,fbLog:=fbLog,byteASCIIBufferToParse:=byteCommandBuffer,byteBinayBufferOutput:=byteADSBuffer);
            ELSE
                bError:=TRUE;
                nErrorID:=701;
                sSubErrorString:='State 6: Buffer index out of range.';
            END_IF
        END_IF;
    ELSE
        bError:=TRUE;
        nErrorId:=fbParseStreamBufferToADS.nErrorId;
        sSubErrorString:='State 6: Failed to parse ASCII buffer to ADS buffer.';
    END_IF;

END_IF

//State 7: Write ADS data
IF (nState=6) THEN
    IF stSymInfo.byteSize>=fbParseStreamBufferToADS.nBinaryBytesWritten THEN //Ensure right size of variable
        fbAdsWriteValue(
            PORT:= nADSPort,
            IDXGRP:= stSymInfo.idxGroup,
            IDXOFFS:= stSymInfo.idxOffset,
            LEN:= fbParseStreamBufferToADS.nBinaryBytesWritten,
            SRCADDR:=ADR(byteADSBuffer[0]) ,
            WRITE:= TRUE,
            TMOUT:= T#5S,
        );
        IF NOT fbAdsWriteValue.ERR THEN
            IF NOT fbAdsWriteValue.BUSY THEN
                fbAdsWriteValue(Write:=FALSE);
                nState:=7;
            END_IF
        ELSE
            bError:=TRUE;
            nErrorId:=fbAdsWriteValue.ERRID;
            sSubErrorString:='State 7: Failed ADS write command.';
        END_IF
    ELSE
            bError:=TRUE;
            nErrorId:=711;
            sSubErrorString:='State 7: Size missmatch between ASCII data and variable size.';
    END_IF
    //fbLog.Error( sMessage := concat(str1:='State 7: ', str2:=PSTRING_TO_STRING(psCommandBufferString)), nErrID := nBytesInCommandBuffer );
END_IF

//State 8: Read data over ADS
IF (((nState=5) AND bReadCmd) OR ((nState=7) AND bWriteCmd AND stSettings.bReturnData)) THEN
    IF(stSymInfo.byteSize>PLCPRJ_BUFFER_SIZE-255) THEN
        nADSBytesToRead:=PLCPRJ_BUFFER_SIZE-255;
    ELSE
        nADSBytesToRead:=stSymInfo.byteSize;
    END_IF
    fbAdsReadValue(
        PORT:= nADSPort,
        IDXGRP:= stSymInfo.idxGroup,
        IDXOFFS:=stSymInfo.idxOffset,
        LEN:= nADSBytesToRead,
        DESTADDR:=ADR(byteADSBuffer),
        Read:= TRUE,
        TMOUT:= T#100MS,
     );

     IF NOT fbAdsReadValue.ERR THEN
        IF NOT fbAdsReadValue.BUSY THEN
            fbAdsReadValue(READ:=FALSE);
            bExecuteWriteBufferToEPICS:=TRUE;
            nState:=8;
        END_IF
    ELSE
        bError:=TRUE;
        nErrorId:=fbAdsReadValue.ERRID;
        sSubErrorString:='State 8: Failed ADS read command.';
    END_IF;
    //fbLog.Error( sMessage := concat(str1:='State 6a: ', str2:=PSTRING_TO_STRING(psCommandBufferString)), nErrID := nBytesInCommandBuffer );
END_IF

//State 9: Parse stream and send to buffer if needed
fbParseADSBufferToStream(bExecute:=bExecuteWriteBufferToEPICS,symbolInfo:=stSymInfo,fbTx:=fbTx,fbLog:=fbLog,byteBufferToSend:=byteADSBuffer,bReturnVariableName:=stSettings.bReturnVarName, sVariableName:=sVariableName, byteFrameBuffer:=byteFrameBuffer,nFrameBufferIndex:=nFrameBufferIndex);
IF (nState=8) THEN
    bExecuteWriteBufferToEPICS:=TRUE;
    IF NOT fbParseADSBufferToStream.bError THEN
        IF NOT fbParseADSBufferToStream.bBusy THEN
            nState:=9;
            bExecuteWriteBufferToEPICS:=FALSE;
        END_IF
    ELSE
        bError:=TRUE;
        nErrorId:=fbParseADSBufferToStream.nErrorId;
        sSubErrorString:='State 9: Failed to parse ADS buffer to ASCII buffer.';
    END_IF
    //fbLog.Error( sMessage := concat(str1:='State 6b: ', str2:=PSTRING_TO_STRING(psCommandBufferString)), nErrID := nBytesInCommandBuffer );
END_IF


//State10: Send data to EPICS
IF ((nState=9) OR ((nState=7) AND NOT stSettings.bReturnData AND bWriteCmd)) THEN
    IF bWriteCmd AND NOT stSettings.bReturnData THEN
        //Copy 'OK' sting to output buffer
        nFrameBufferIndex:=len(STR:=EPICS_ACK_STRING);
        memcpy(destAddr:=ADR(byteFrameBuffer[0]),srcAddr:=ADR(EPICS_ACK_STRING), nFrameBufferIndex);
    ELSIF bReadCmd OR stSettings.bReturnData THEN
        IF nFrameBufferIndex> EPICS_MAX_FRAME_SIZE-3 THEN  //must be space for atleast 3 bytes  (';crlf')
            fbTx.AddTail( bPut := ADR(byteFrameBuffer[0]), nWriteCount:=nFrameBufferIndex );(* Put string to the tx fifo *)
            IF NOT fbTx.bOk THEN(* TX fifo overflow => log error *)
                bError:=TRUE;
                nErrorId:=801;
                sSubErrorString:='State 7c: TX buffer overflow.';
            END_IF
            nFrameBufferIndex:=0;
        END_IF
    END_IF;
    nCleanBytes:=0;
    //check for semi-colon and add it to output buffer
    IF(byteCommandBuffer[nIndexEndOfCommand]=F_ToASC(str:=EPICS_COMMAND_DELIMITER)) THEN //CR or LF
        byteFrameBuffer[nFrameBufferIndex]:=byteCommandBuffer[nIndexEndOfCommand];
        nFrameBufferIndex:=nFrameBufferIndex+1;
        nCleanBytes:=nCleanBytes+1;
        IF(byteCommandBuffer[nIndexEndOfCommand+1]=EPICS_ASCII_LN OR byteCommandBuffer[nIndexEndOfCommand+1]=EPICS_ASCII_CR) THEN //CR or LF
            byteFrameBuffer[nFrameBufferIndex]:=byteCommandBuffer[nIndexEndOfCommand+1];
            nFrameBufferIndex:=nFrameBufferIndex+1;
            nCleanBytes:=nCleanBytes+1;
        END_IF;
        IF(byteCommandBuffer[nIndexEndOfCommand+2]=EPICS_ASCII_LN OR byteCommandBuffer[nIndexEndOfCommand+2]=EPICS_ASCII_CR) THEN //CR or LF
            byteFrameBuffer[nFrameBufferIndex]:=byteCommandBuffer[nIndexEndOfCommand+2];
            nFrameBufferIndex:=nFrameBufferIndex+1;
            nCleanBytes:=nCleanBytes+1;
        END_IF;

        //Send OK or data to output queue
        fbTx.AddTail( bPut := ADR(byteFrameBuffer[0]), nWriteCount:=nFrameBufferIndex );(* Put string to the tx fifo *)
        IF NOT fbTx.bOk THEN(* TX fifo overflow => log error *)
            bError:=TRUE;
            nErrorId:=802;
            sSubErrorString:='State 8: TX buffer overflow.';
        ELSE
            nState:=10;
        END_IF
    ELSE
            bError:=TRUE;
            nErrorId:=803;
            sSubErrorString:='State 8: Semi-colon missing.';
    END_IF
    //fbLog.Error( sMessage := concat(str1:='State : ', str2:=PSTRING_TO_STRING(psCommandBufferString)), nErrID := nBytesInCommandBuffer );
END_IF


//State 11: Clean ";" and CR or LN from buffer, also see if extra zeros(=0) in buffer..
IF (nState=10) THEN
    IF nCleanBytes>0 THEN
        F_RemoveBytesFromBuffer(nCleanBytes,byteCommandBuffer:=byteCommandBuffer,nBytesInCommandBuffer:=nBytesInCommandBuffer,nIndexEndOfCommand:=nIndexEndOfCommand);
    END_IF;
    //Clean extra bytes/spaces Check if extra empty bytes
    iEmptyCounter:=0;
    IF nBytesInCommandBuffer>0 THEN
        WHILE byteCommandBuffer[iEmptyCounter]=0 AND iEmptyCounter<nBytesInCommandBuffer DO
            iEmptyCounter:=iEmptyCounter+1;
        END_WHILE
        //remove bytes
        F_RemoveBytesFromBuffer(iEmptyCounter,byteCommandBuffer:=byteCommandBuffer,nBytesInCommandBuffer:=nBytesInCommandBuffer,nIndexEndOfCommand:=nIndexEndOfCommand);
    END_IF

    nState:=11;
    //fbLog.Error( sMessage := concat(str1:='State 8: ', str2:=PSTRING_TO_STRING(psCommandBufferString)), nErrID := nBytesInCommandBuffer );
END_IF

// Command ready: Start over
IF (nState=11) THEN
    nState:=0;
    bReadCmd:=FALSE;
    bWriteCmd:=FALSE;
    nIndexEndOfCommand:=0;
    bExecuteWriteBufferToEPICS:=FALSE;
    //fbLog.Error( sMessage := concat(str1:='State 9: ', str2:=PSTRING_TO_STRING(psCommandBufferString)), nErrID := nBytesInCommandBuffer );
    IF nBytesInCommandBuffer<0 THEN
        nBytesInCommandBuffer:=0;
    END_IF
    fbAdsReadValue(read:=FALSE);
    fbAdsWriteValue(WRITE:=FALSE);
    fbSymInfoByName(start:=FALSE);

END_IF

//Ensure that communiucation not hangs du to stuck in one state

fbStateTimoutTimer(In:=(nState>0 OR nBytesInCommandBuffer>0), PT:=EPICS_COM_TIMEOUT);
IF fbStateTimoutTimer.Q THEN //latch in in which state stucked

    nErrorID:=nState*10;
    IF nBytesInCommandBuffer>0 THEN
        nErrorID:=1;
    END_IF
    sSubErrorString:='State timout. To long time in one state.';
    bError:=TRUE;
    //Latch buffer at error
    MEMCPY(destAddr:=ADR(sComBufferAtError[0]),srcAddr:=ADR(byteCommandBuffer[0]),n:=255); //For debug purpose
    fbLog.Error( sMessage := 'State timeout', nErrID := nErrorID );
    fbAdsReadValue(read:=FALSE);
    fbAdsWriteValue(WRITE:=FALSE);
    fbSymInfoByName(start:=FALSE);
END_IF

//Send error message to host
IF bError AND NOT bErrorOld  THEN
    nErrorCounter:=nErrorCounter+1;
    sError:=concat(str1:='Error ', STR2:=UDINT_TO_STRING(nErrorID));
    sError:=CONCAT(str1:=sError , STR2:=' : ');
    sError:=CONCAT(str1:=sError , STR2:=sSubErrorString);
    sError:=CONCAT(str1:=sError , STR2:='  ');
    nLength:=len(STR:=sError);
    sError[nLength-2]:=EPICS_ASCII_COMMAND_DELIMITER;
    sError[nLength-1]:=10; //LF
    fbLog.Error( sMessage := sError, nErrID := nErrorID );
    fbTx.AddTail( bPut :=ADR(sError) , nWriteCount:=nLength);(* Put string to the tx fifo *)
    IF NOT fbTx.bOk THEN(* TX fifo overflow => log error *)
        bError:=TRUE;
        fbLog.Error( sMessage := 'TX overflow ', nErrID := nErrorId );
    END_IF
    bErrorMessageSent:=TRUE;
END_IF

IF  bReset OR fbStateTimoutTimer.Q THEN
    fbStateTimoutTimer(In:=FALSE);
    nState:=0;
    bReadCmd:=FALSE;
    bWriteCmd:=FALSE;
    //Clear buffer
    nIndexEndOfCommand:=0;
    MEMSET(ADR(byteCommandBuffer),0,SIZEOF(byteCommandBuffer));
    nBytesInCommandBuffer:=0;
    bExecuteWriteBufferToEPICS:=FALSE;
    bErrorMessageSent:=FALSE;
    nErrorId:=0;
    bError:=0;
END_IF
bErrorOld:=bError;

END_FUNCTION_BLOCK

// ---- POUs/Helper POUs/FB_FrameFifo.TcPOU
(* Tx (byte data) fifo control function block (Older where based on string format) *)
FUNCTION_BLOCK FB_FrameFifo
VAR
    sVersion: STRING:='0.9.0';
END_VAR
VAR_INPUT
    bLog        : BOOL          := FALSE;(* TRUE => Enable log message output, FALSE => Disable *)
    sPrefix     : STRING        := 'Unknown::';(* Log message description string (allows the identification of log message source) *)
    bPut        : POINTER TO ARRAY[0..EPICS_MAX_FRAME_SIZE] OF BYTE; (* Byte message to add (write) to the fifo *)
    bGet        : POINTER TO ARRAY[0..EPICS_MAX_FRAME_SIZE] OF BYTE; (* Byte message removed (read) from fifo *)
    nWriteCount : UDINT:=0;
    nReadBufferSize : UDINT:=0;
END_VAR
VAR_OUTPUT
    bOk         : BOOL;         (* TRUE = New entry added or removed succesfully, FALSE = Fifo overflow or fifo empty *)
    nCount      : UDINT         := 0;(* Number of fifo entries *)
    cbFree      : UDINT         := 0;(* Free buffer space *)
    nReadCount  : UDINT:=0;
END_VAR
VAR
    fbBuffer    : FB_MemRingBuffer;(* Basic (lower level) string buffer control function block *)
    buffer      : ARRAY[-3..PLCPRJ_BUFFER_SIZE] OF BYTE;(* Internal buffer memory *)
    sPut        : T_MaxString;
    nMax: UDINT;
    spBufferString: POINTER TO STRING;
END_VAR



;

ACTION Clear:
(* Resets fifo = clears all data *)
fbBuffer.A_Reset( pBuffer:= ADR(buffer), cbBuffer:= SIZEOF(buffer),
                bOk=>bOk, nCount=>nCount );
cbFree := PLCPRJ_BUFFER_SIZE;(* Free buffer size *)
END_ACTION

ACTION AddTail:
(* Adds new fifo entry *)
fbBuffer.A_AddTail( pBuffer:= ADR(buffer),pWrite:=bPut,cbWrite:=nWriteCount,cbBuffer:= SIZEOF(buffer),
                     bOk=>bOk, nCount=>nCount );

IF bOk THEN
    cbFree := PLCPRJ_BUFFER_SIZE - fbBuffer.cbSize;(* Calculate the free buffer space *)
    IF bLog THEN(* Log message *)
        IF  nWriteCount>50 THEN
            nMax:=50;
        ELSE
            nMax:=nWriteCount;
        END_IF
        sPut:='';
        memcpy(destAddr:=ADR(sPut[0]),srcAddr:=(bPut+nWriteCount-nMax),n:=nMax); //Copy byte data to string
        sPut[nMax]:=0; //Terminate string
        ADSLOGSTR( ADSLOG_MSGTYPE_HINT OR ADSLOG_MSGTYPE_LOG, CONCAT( ''(*sPrefix*), '"%s"' ),sPut );
    END_IF
END_IF
END_ACTION

ACTION RemoveHead:
(* Removes oldest fifo entry *)
//fbBuffer.A_RemoveHead( pBuffer:= ADR(buffer), cbBuffer:= SIZEOF(buffer), pRead:=bGet,
//                      bOk=>bOk,cbReturn=>nReadCount, nCount=>nCount, cbRead:=nReadBufferSize);
fbBuffer.A_RemoveHead( pBuffer:= ADR(buffer), cbBuffer:= SIZEOF(buffer), pRead:=bGet,
                        bOk=>bOk,cbReturn=>nReadCount, nCount=>nCount, cbRead:=nReadBufferSize);



IF bOk THEN
    cbFree := PLCPRJ_BUFFER_SIZE - fbBuffer.cbSize;(* Calculate the free buffer space *)
    //ADSLOGSTR( ADSLOG_MSGTYPE_HINT OR ADSLOG_MSGTYPE_LOG, CONCAT( 'Took bytes OK: ', '"%s"' ) ,UDINT_TO_STRING(ncount));
ELSE

    //ADSLOGSTR( ADSLOG_MSGTYPE_HINT OR ADSLOG_MSGTYPE_LOG, CONCAT( ''(*sPrefix*), '"%s"' ),'Took bytes Fail' );
END_IF
END_ACTION

END_FUNCTION_BLOCK

// ---- POUs/Helper POUs/FB_LogFifo.TcPOU
(* Log/debug/error message fifo *)
FUNCTION_BLOCK FB_LogFifo
VAR
    sVersion: STRING:='0.9.0';
END_VAR
VAR_INPUT
    bLog        : BOOL      := FALSE;(* TRUE => Enable log message output, FALSE => Disable *)
    sPrefix     : STRING    := 'Unknown::';(* Log message description string (allows the identification of log message source) *)

    sMessage    : STRING    := '';(* String message to add (write) to the fifo *)
    nErrID      : UDINT     := 0;(* Error code to add (write) to the fifo *)
    hSocket     : T_HSOCKET;(* Socket connection handle *)
END_VAR
VAR_OUTPUT
    bOk         : BOOL;(* TRUE = New entry added or removed succesfully, FALSE = Fifo overflow or fifo empty *)
    sGet        : T_MaxString := '';(* String entry removed (read) from fifo *)
    nCount      : UDINT := 0;(* Number of fifo entries *)
END_VAR
VAR
    fbBuffer    : FB_StringRingBuffer;(* Basic (lower level) string buffer control function block *)
    buffer      : ARRAY[0..PLCPRJ_BUFFER_SIZE] OF BYTE;(* Internal buffer memory *)
    sSource     : T_MaxString;
    sPut        : T_MaxString;
END_VAR

;

ACTION Clear:
(* Clears all fifo entries *)
fbBuffer.A_Reset(   pBuffer := ADR( buffer ), cbBuffer := SIZEOF( buffer ),
                    bOk=>bOk, nCount=>nCount, getValue=>sGet );
END_ACTION

ACTION Error:
(* Adds new fifo entry *)

IF nErrID = 0 THEN
    sSource := '::Error: 0x';
ELSIF ( nErrID AND 16#80000000) = 16#80000000 THEN
    IF nErrID = 16#80072746 THEN
        sSource := '::Win32 error (the connection is reset by remote side): 0x';
    ELSE
        sSource := '::Win32 error: 0x';
    END_IF
ELSIF (nErrID AND 16#00008100) = 16#00008100 THEN
    CASE nErrID OF
        PLCPRJ_ERROR_RECEIVE_TIMEOUT:
            sSource := '::PLC sample project receive timeout error: 0x';
        PLCPRJ_ERROR_SENDFIFO_OVERFLOW:
            sSource := '::PLC sample project send fifo overflow error: 0x';
        PLCPRJ_ERROR_RECFIFO_OVERFLOW:
            sSource := '::PLC sample project receive fifo overflow error: 0x';
    ELSE
        sSource := '::Other PLC sample project error: 0x';
    END_CASE
ELSIF (nErrID AND 16#00008000) = 16#00008000 THEN
    sSource := '::Internal TCP/IP Connection Server error: 0x';
ELSE
    sSource := '::TwinCAT System error: 0x';
END_IF

sPut := CONCAT( CONCAT( CONCAT( sPrefix, sMessage ), sSource ), DWORD_TO_HEXSTR( nErrID AND 16#FFFF, 0, FALSE ) );

fbBuffer.A_AddTail( pBuffer:= ADR(buffer), cbBuffer:= SIZEOF(buffer),
                    putValue:= sPut, bOk=>bOk, nCount=>nCount );
IF bOk THEN
    IF bLog THEN(* Log error message *)
        ADSLOGSTR( ADSLOG_MSGTYPE_ERROR OR ADSLOG_MSGTYPE_LOG, '%s', sPut );
    END_IF
END_IF
END_ACTION

ACTION Remove:
(* Removes oldest fifo entry *)
IF nCount = 0 THEN
    sGet := '';
    bOk := FALSE;
    RETURN;
END_IF

fbBuffer.A_RemoveHead( pBuffer:= ADR(buffer), cbBuffer:= SIZEOF(buffer),
                        getValue=>sGet, bOk=>bOk, nCount=>nCount );
END_ACTION

ACTION Message:
(* Adds new fifo entry *)

sPut := CONCAT( CONCAT( sPrefix, sMessage ), CONCAT( '::', HSOCKET_TO_STRING(hSocket) ) );
fbBuffer.A_AddTail( pBuffer:= ADR(buffer), cbBuffer:= SIZEOF(buffer),
                    putValue:= sPut, bOk=>bOk, nCount=>nCount );
IF bOk THEN
    IF bLog THEN(* Log information message *)
        ADSLOGSTR( ADSLOG_MSGTYPE_HINT OR ADSLOG_MSGTYPE_LOG, '%s', sPut );
    END_IF
END_IF
END_ACTION

END_FUNCTION_BLOCK

// ---- POUs/FB_ADSBufferToStreamBuffer.TcPOU
///#########################################################
///Function block used to convert binary ADS buffer to ASCII Stream buffer
/// Library:
///
///
/// Global Variables:
/// - EPICS_MAX_FRAME_SIZE
/// - EPICS_ARRAY_DELIMITER
/// - EPICS_COMMAND_DELIMITER
/// - PLCPRJ_BUFFER_SIZE
///
/// Data types:
///
/// External functions:
///     - TC2_Standard lib
///     - Tc2_Utilities lib
///     - Tc2_System lib
///
///###########################################################

FUNCTION_BLOCK FB_ADSBufferToStreamBuffer
VAR
    sVersion: STRING:='0.9.0';
END_VAR
VAR_INPUT
    bExecute: BOOL;
    symbolInfo:SYMINFOSTRUCT;
    sVariableName:STRING:='';
    bReturnVariableName:BOOL:=FALSE;
END_VAR
VAR_IN_OUT
    fbTx        : FB_FrameFifo;(* TX fifo * To send *)
    fbLog       : FB_LogFifo;(* Log message fifo *)
    byteBufferToSend    : ARRAY[0..PLCPRJ_BUFFER_SIZE] OF BYTE;
    byteFrameBuffer: ARRAY[0..EPICS_MAX_FRAME_SIZE] OF BYTE;
    nFrameBufferIndex:INT:=0;
END_VAR

VAR
    nADSBytesToRead:INT:=0;
    nSize: INT;
    i: INT;
    sTemp: STRING(255):='';
    nErrorCode:UDINT;
    //Below data types are supported by the EPCIS interface
    pINT16 :POINTER TO INT;
    pBYTE8: POINTER TO BYTE;
    pSINT8: POINTER TO SINT;
    pUINT16:POINTER TO UINT;
    pINT32: POINTER TO DINT;
    pUINT32:POINTER TO UDINT;
    pLINT64:POINTER TO LINT;
    pULINT64:POINTER TO ULINT;
    pREAL32:POINTER TO REAL;
    pREAL64:POINTER TO LREAL;
    pBOOL: POINTER TO BOOL;
    pString: POINTER TO STRING;


    //ADS_BIG types (structs)
    fbReadDUT_AxisStatus_v0_01:FB_Read_DUT_AxisStatus_v0_01;

    //Buffer to push data into Frame Buffer
    pbEpicsCommandDelimiter: POINTER TO BYTE;
    iADSReadBufferIndex: INT;
    bTransferInASCII: BOOL:=TRUE; //Otherwise binary format
    nBytes: INT;
    //fArray:POINTER TO ARRAY[0..10] OF LREAL;
    bExecuteOld: BOOL:=FALSE;
    sValue: STRING;
    nCompensation: INT;
END_VAR

VAR_OUTPUT
    bBusy: BOOL:=FALSE;
    bDone: BOOL:=FALSE;
    bError: BOOL:=FALSE;
    nErrorId: UDINT:=0;
    bADSToFrameBufferComplete: BOOL;
END_VAR




bBusy:=TRUE;
bDone:=FALSE;
bError:=FALSE;

//prepare for new command
IF NOT bExecuteOld AND bExecute THEN
    iADSReadBufferIndex:=0;
    bADSToFrameBufferComplete:=FALSE;
END_IF

IF bExecute THEN
    nFrameBufferIndex:=0;
    IF(symbolInfo.byteSize>PLCPRJ_BUFFER_SIZE) AND iADSReadBufferIndex=0 THEN
        nADSBytesToRead:=UDINT_TO_INT(PLCPRJ_BUFFER_SIZE);
    ELSE
        nADSBytesToRead:=UDINT_TO_INT( symbolInfo.byteSize);
    END_IF
    IF bReturnVariableName THEN //Include variablename in string to return to EPCIS
        nFrameBufferIndex:=len(sVariableName);
        MEMCPY(destAddr:=ADR(byteFrameBuffer[0]),srcAddr:=ADR(sVariableName),n:=nFrameBufferIndex);
        byteFrameBuffer[nFrameBufferIndex]:=EPICS_ASCII_EQUAL;
        nFrameBufferIndex:=nFrameBufferIndex+1;
    END_IF
    IF NOT (symbolInfo.adsDataType= ADST_STRING OR  symbolInfo.adsDataType=ADST_BIGTYPE OR  symbolInfo.adsDataType=ADST_WSTRING OR symbolInfo.adsDataType=ADST_MAXTYPES OR symbolInfo.adsDataType=ADST_REAL80  OR symbolInfo.adsDataType=ADST_VOID) THEN
        nErrorId:=0;
        bADSToFrameBufferComplete:=TRUE;
        CASE symbolInfo.adsDataType OF
            ADST_INT8: //sint
                nSize:=1;
                nCompensation:=1;
            ADST_UINT8:  //byte
                nSize:=1;
                nCompensation:=1;
            ADST_INT16:
                nSize:=2;
                nCompensation:=1;
            ADST_UINT16:
                nSize:=2;
                nCompensation:=1;
            ADST_INT32:  //Dint
                nSize:=4;
                nCompensation:=2;
            ADST_UINT32:
                nSize:=4;
                nCompensation:=2;
            ADST_INT64:
                nSize:=8;
                nCompensation:=2;
            ADST_UINT64:
                nSize:=8;
                nCompensation:=2;
            ADST_REAL32:
                nSize:=4;
                nCompensation:=2;
            ADST_REAL64:
                nSize:=8;
                nCompensation:=2;
            ADST_BIT:
                nSize:=1;
                nCompensation:=1;
        END_CASE
        FOR i:=iADSReadBufferIndex TO (nADSBytesToRead-nCompensation) BY nSize DO

            CASE symbolInfo.adsDataType OF
                ADST_INT8: //sint
                    nSize:=1;
                    pSINT8:=ADR(byteBufferToSend[i]);
                    sTemp:=SINT_TO_STRING( Tc2_Utilities.PSINT_TO_SINT(pSINT8));
                ADST_UINT8:  //byte
                    nSize:=1;
                    pBYTE8:=ADR(byteBufferToSend[i]);
                    sTemp:=BYTE_TO_STRING( Tc2_Utilities.PBYTE_TO_BYTE(pBYTE8));
                ADST_INT16:
                    nSize:=2;
                    pInt16:=ADR(byteBufferToSend[i]);
                    sTemp:=INT_TO_STRING( Tc2_Utilities.PINT_TO_INT(pInt16));
                ADST_UINT16:
                    nSize:=2;
                    puInt16:=ADR(byteBufferToSend[i]);
                    sTemp:=INT_TO_STRING( Tc2_Utilities.PUINT_TO_UINT(puInt16));
                ADST_INT32:  //Dint
                    nSize:=4;
                    pInt32:=ADR(byteBufferToSend[i]);
                    sTemp:=DINT_TO_STRING( Tc2_Utilities.PDINT_TO_DINT(pInt32));
                ADST_UINT32:
                    nSize:=4;
                    puInt32:=ADR(byteBufferToSend[i]);
                    sTemp:=UDINT_TO_STRING( Tc2_Utilities.PUDINT_TO_UDINT(puInt32));
                ADST_INT64:
                    nSize:=8;
                    pLINT64:=ADR(byteBufferToSend[i]);
                    sTemp:=LINT_TO_STRING( Tc2_Utilities.PLINT_TO_LINT(pLINT64));
                ADST_UINT64:
                    nSize:=8;
                    pULINT64:=ADR(byteBufferToSend[i]);
                    sTemp:=ULINT_TO_STRING( Tc2_Utilities.PULINT_TO_ULINT(pULINT64));
                ADST_REAL32:
                    nSize:=4;
                    pREAL32:=ADR(byteBufferToSend[i]);
                    sTemp:=REAL_TO_STRING( Tc2_Utilities.PREAL_TO_REAL(pREAL32));
                ADST_REAL64: //LREAL
                    nSize:=8;
                    pREAL64:=ADR(byteBufferToSend[i]);
                    sTemp:=LREAL_TO_STRING( Tc2_Utilities.PLREAL_TO_LREAL(pREAL64));
                ADST_BIT:
                    nSize:=1;
                    pBOOL:=ADR(byteBufferToSend[i]);
                    IF Tc2_Utilities.PBOOL_TO_BOOL(pBOOL)THEN
                        sTemp:='1';
                    ELSE
                        sTemp:='0';
                    END_IF
            END_CASE

            IF i>0 THEN // dont and separator for first value
                sTemp:=Tc2_Standard.CONCAT(str1:=EPICS_ARRAY_DELIMITER,str2:=sTemp);
            END_IF;
            IF (nFrameBufferIndex+len(sTemp)+3)>EPICS_MAX_FRAME_SIZE THEN
                fbTx.AddTail( bPut := ADR(byteFrameBuffer), nWriteCount:=nFrameBufferIndex );(* Put string to the tx fifo *)
                nFrameBufferIndex:=0;

                IF NOT fbTx.bOk THEN(* TX fifo overflow => log error *)
                    fbLog.Error( sMessage := 'FB_FrameFifo(sender)', nErrID := PLCPRJ_ERROR_SENDFIFO_OVERFLOW );
                    bError:=TRUE;
                    nErrorId:=PLCPRJ_ERROR_SENDFIFO_OVERFLOW;
                    RETURN;
                END_IF
                iADSReadBufferIndex:=i;
                bADSToFrameBufferComplete:=FALSE;
                EXIT; //One frame is full wait untill sent then contiue for loop to fill next frame
            ELSE
                memcpy(srcAddr:=ADR(sTemp),destAddr:=ADR(byteFrameBuffer)+nFrameBufferIndex,n:=len(sTemp));
                nFrameBufferIndex:=nFrameBufferIndex+len(sTemp);
            END_IF
        END_FOR;
    ELSE
        CASE symbolInfo.adsDataType OF
                ADST_VOID:
                    ; //Data type ADST_VOID not implmented
                ADST_STRING:
                    pString:=ADR(byteBufferToSend[0]);
                    nFrameBufferIndex:=nFrameBufferIndex+MIN(nADSBytesToRead,len(STR :=PSTRING_TO_STRING(pString)));//Find length of string
                    memcpy(srcAddr:=ADR(byteBufferToSend[0]),destAddr:=ADR(byteFrameBuffer[0]),n:=nFrameBufferIndex);
                    bADSToFrameBufferComplete:=TRUE;
                ADST_WSTRING:
                    ; //Data type ADST_WSTRING not implmented
                ADST_BIGTYPE:
                    //Support for structures (DUT)
                    //Add FB:s generated by TwinCatEpicsUtilities here (also needs to be declared)
                    fbReadDUT_AxisStatus_v0_01(sVariableName:=sVariableName,sSymDataType:=symbolInfo.symDataType,byteADSReadBuffer:=byteBufferToSend,byteFrameBuffer:=byteFrameBuffer,fbTx:=fbTx,fbLog:=fbLog,iFrameBufferIndex:=nFrameBufferIndex,bReady:=bADSToFrameBufferComplete);
                ADST_MAXTYPES:
                    ; //Data type ADST_MAXTYPES not implmented
                ADST_REAL80:
                    ; //Data type ADST_REAL80 not implmented1
        END_CASE
    END_IF
    //Terminate and go to next step if ADS buffer is empty, otherwise execute this state once more.
    IF bADSToFrameBufferComplete (*AND nFrameBufferIndex > 0 *) THEN
    (*  //Add end delimiters, last string
        pbEpicsCommandDelimiter:=ADR(EPICS_COMMAND_DELIMITER);
        byteFrameBuffer[nFrameBufferIndex]:=  PBYTE_TO_BYTE(pbEpicsCommandDelimiter);
        nFrameBufferIndex:=nFrameBufferIndex+1;
        IF bWriteFrameTerminator THEN
            byteFrameBuffer[nFrameBufferIndex]:=byteTerminator;     //LN or CR
            nFrameBufferIndex:=nFrameBufferIndex+1;                 //Buffer starts from 0
        END_IF

        fbTx.AddTail( bPut := ADR(byteFrameBuffer[0]), nWriteCount:=nFrameBufferIndex);(* Put string to the tx fifo *)
        IF NOT fbTx.bOk THEN(* TX fifo overflow => log error *)
            fbLog.Error( sMessage := 'FB_FrameFifo(sender)', nErrID := PLCPRJ_ERROR_SENDFIFO_OVERFLOW );
            bError:=TRUE;
            nErrorId:=PLCPRJ_ERROR_SENDFIFO_OVERFLOW;
            RETURN;
        END_IF
        bADSToFrameBufferComplete:=FALSE;*)
        bBusy:=FALSE;
        bDone:=TRUE;
    END_IF
ELSE
    bBusy:=FALSE;
    bDone:=FALSE;
    bError:=FALSE;
    nErrorId:=0;
    bADSToFrameBufferComplete:=FALSE;
END_IF
bExecuteOld:=bExecute;

END_FUNCTION_BLOCK

// ---- POUs/DUT_Support/FB_Read_DUT_AxisStatus_v0_01.TcPOU
FUNCTION_BLOCK FB_Read_DUT_AxisStatus_v0_01
VAR_INPUT
    sVariableName:STRING;
    sSymDataType:STRING;
END_VAR
VAR
    pInputDataBuffer    :   POINTER TO DUT_AxisStatus_v0_01;
    iCounter            :   INT:=0;
    sValue              :   STRING;
    iLength             :   INT:=0;
END_VAR
VAR_IN_OUT
    byteADSReadBuffer   :   ARRAY[0..PLCPRJ_BUFFER_SIZE] OF BYTE;//ADS input buffer
    byteFrameBuffer     :   ARRAY[0..EPICS_MAX_FRAME_SIZE] OF BYTE;
    fbTx                :   FB_FrameFifo;// TX fifo * To send
    fbLog               :   FB_LogFifo;// Log message fifo
    bReady              :   BOOL; //Allways transfer stucts in the same frame (max size is 1500byte)
    iFrameBufferIndex   :   INT;
END_VAR


IF find(STR1:=sSymDataType,STR2:='DUT_AxisStatus_v0_01')>0 THEN
    iFrameBufferIndex:=0;
    iCounter:=iCounter+1; //Just to see execution
    pInputDataBuffer:=ADR(byteADSReadBuffer);//ADR(bADSReadBuffer[0]);
    //Add variable name to output frame
    iLength:=len(str:=sVariableName);
    memcpy(srcAddr:=ADR(sVariableName),destAddr:=ADR(byteFrameBuffer[iFrameBufferIndex]),n:=iLength);
    iFrameBufferIndex:=iFrameBufferIndex+iLength;
    byteFrameBuffer[iFrameBufferIndex]:=EPICS_ASCII_EQUAL;  // =

    iFrameBufferIndex:=iFrameBufferIndex+1;

    IF pInputDataBuffer^.bEnable THEN
        byteFrameBuffer[iFrameBufferIndex]:=EPICS_ASCII_ONE; // 1
    ELSE
        byteFrameBuffer[iFrameBufferIndex]:=EPICS_ASCII_ZERO; // 0
    END_IF
    iFrameBufferIndex:=iFrameBufferIndex+1;
    byteFrameBuffer[iFrameBufferIndex]:=EPICS_ASCII_COMMA; // ,
    iFrameBufferIndex:=iFrameBufferIndex+1;

        IF iFrameBufferIndex>=EPICS_MAX_FRAME_SIZE-25 THEN  //Send before full buffer
            fbTx.AddTail( bPut := ADR(byteFrameBuffer), nWriteCount:=iFrameBufferIndex);(* Put string to the tx fifo *)
            IF NOT fbTx.bOk THEN(* TX fifo overflow => log error *)
             fbLog.Error( sMessage := 'FB_FrameFifo(sender)', nErrID := PLCPRJ_ERROR_SENDFIFO_OVERFLOW );
            END_IF
            iFrameBufferIndex:=0;
        END_IF

    IF pInputDataBuffer^.bReset THEN
        byteFrameBuffer[iFrameBufferIndex]:=EPICS_ASCII_ONE; // 1
    ELSE
        byteFrameBuffer[iFrameBufferIndex]:=EPICS_ASCII_ZERO; // 0
    END_IF
    iFrameBufferIndex:=iFrameBufferIndex+1;
    byteFrameBuffer[iFrameBufferIndex]:=EPICS_ASCII_COMMA; // ,
    iFrameBufferIndex:=iFrameBufferIndex+1;

        IF iFrameBufferIndex>=EPICS_MAX_FRAME_SIZE-25 THEN  //Send before full buffer
            fbTx.AddTail( bPut := ADR(byteFrameBuffer), nWriteCount:=iFrameBufferIndex);(* Put string to the tx fifo *)
            IF NOT fbTx.bOk THEN(* TX fifo overflow => log error *)
             fbLog.Error( sMessage := 'FB_FrameFifo(sender)', nErrID := PLCPRJ_ERROR_SENDFIFO_OVERFLOW );
            END_IF
            iFrameBufferIndex:=0;
        END_IF

    IF pInputDataBuffer^.bExecute THEN
        byteFrameBuffer[iFrameBufferIndex]:=EPICS_ASCII_ONE; // 1
    ELSE
        byteFrameBuffer[iFrameBufferIndex]:=EPICS_ASCII_ZERO; // 0
    END_IF
    iFrameBufferIndex:=iFrameBufferIndex+1;
    byteFrameBuffer[iFrameBufferIndex]:=EPICS_ASCII_COMMA; // ,
    iFrameBufferIndex:=iFrameBufferIndex+1;

        IF iFrameBufferIndex>=EPICS_MAX_FRAME_SIZE-25 THEN  //Send before full buffer
            fbTx.AddTail( bPut := ADR(byteFrameBuffer), nWriteCount:=iFrameBufferIndex);(* Put string to the tx fifo *)
            IF NOT fbTx.bOk THEN(* TX fifo overflow => log error *)
             fbLog.Error( sMessage := 'FB_FrameFifo(sender)', nErrID := PLCPRJ_ERROR_SENDFIFO_OVERFLOW );
            END_IF
            iFrameBufferIndex:=0;
        END_IF

    sValue:= UINT_TO_STRING(pInputDataBuffer^.nCommand);
    iLength:=len(str:=sValue);
    memcpy(srcAddr:=ADR(sValue),destAddr:=ADR(byteFrameBuffer[iFrameBufferIndex]),n:=iLength);
    iFrameBufferIndex:=iFrameBufferIndex+iLength;
    byteFrameBuffer[iFrameBufferIndex]:=EPICS_ASCII_COMMA; // ,
    iFrameBufferIndex:=iFrameBufferIndex+1;

        IF iFrameBufferIndex>=EPICS_MAX_FRAME_SIZE-25 THEN  //Send before full buffer
            fbTx.AddTail( bPut := ADR(byteFrameBuffer), nWriteCount:=iFrameBufferIndex);(* Put string to the tx fifo *)
            IF NOT fbTx.bOk THEN(* TX fifo overflow => log error *)
             fbLog.Error( sMessage := 'FB_FrameFifo(sender)', nErrID := PLCPRJ_ERROR_SENDFIFO_OVERFLOW );
            END_IF
            iFrameBufferIndex:=0;
        END_IF

    sValue:= UINT_TO_STRING(pInputDataBuffer^.nCmdData);
    iLength:=len(str:=sValue);
    memcpy(srcAddr:=ADR(sValue),destAddr:=ADR(byteFrameBuffer[iFrameBufferIndex]),n:=iLength);
    iFrameBufferIndex:=iFrameBufferIndex+iLength;
    byteFrameBuffer[iFrameBufferIndex]:=EPICS_ASCII_COMMA; // ,
    iFrameBufferIndex:=iFrameBufferIndex+1;

        IF iFrameBufferIndex>=EPICS_MAX_FRAME_SIZE-25 THEN  //Send before full buffer
            fbTx.AddTail( bPut := ADR(byteFrameBuffer), nWriteCount:=iFrameBufferIndex);(* Put string to the tx fifo *)
            IF NOT fbTx.bOk THEN(* TX fifo overflow => log error *)
             fbLog.Error( sMessage := 'FB_FrameFifo(sender)', nErrID := PLCPRJ_ERROR_SENDFIFO_OVERFLOW );
            END_IF
            iFrameBufferIndex:=0;
        END_IF

    sValue:= LREAL_TO_STRING(pInputDataBuffer^.fVelocity);
    iLength:=len(str:=sValue);
    memcpy(srcAddr:=ADR(sValue),destAddr:=ADR(byteFrameBuffer[iFrameBufferIndex]),n:=iLength);
    iFrameBufferIndex:=iFrameBufferIndex+iLength;
    byteFrameBuffer[iFrameBufferIndex]:=EPICS_ASCII_COMMA; // ,
    iFrameBufferIndex:=iFrameBufferIndex+1;

        IF iFrameBufferIndex>=EPICS_MAX_FRAME_SIZE-25 THEN  //Send before full buffer
            fbTx.AddTail( bPut := ADR(byteFrameBuffer), nWriteCount:=iFrameBufferIndex);(* Put string to the tx fifo *)
            IF NOT fbTx.bOk THEN(* TX fifo overflow => log error *)
             fbLog.Error( sMessage := 'FB_FrameFifo(sender)', nErrID := PLCPRJ_ERROR_SENDFIFO_OVERFLOW );
            END_IF
            iFrameBufferIndex:=0;
        END_IF

    sValue:= LREAL_TO_STRING(pInputDataBuffer^.fPosition);
    iLength:=len(str:=sValue);
    memcpy(srcAddr:=ADR(sValue),destAddr:=ADR(byteFrameBuffer[iFrameBufferIndex]),n:=iLength);
    iFrameBufferIndex:=iFrameBufferIndex+iLength;
    byteFrameBuffer[iFrameBufferIndex]:=EPICS_ASCII_COMMA; // ,
    iFrameBufferIndex:=iFrameBufferIndex+1;

        IF iFrameBufferIndex>=EPICS_MAX_FRAME_SIZE-25 THEN  //Send before full buffer
            fbTx.AddTail( bPut := ADR(byteFrameBuffer), nWriteCount:=iFrameBufferIndex);(* Put string to the tx fifo *)
            IF NOT fbTx.bOk THEN(* TX fifo overflow => log error *)
             fbLog.Error( sMessage := 'FB_FrameFifo(sender)', nErrID := PLCPRJ_ERROR_SENDFIFO_OVERFLOW );
            END_IF
            iFrameBufferIndex:=0;
        END_IF

    sValue:= LREAL_TO_STRING(pInputDataBuffer^.fAcceleration);
    iLength:=len(str:=sValue);
    memcpy(srcAddr:=ADR(sValue),destAddr:=ADR(byteFrameBuffer[iFrameBufferIndex]),n:=iLength);
    iFrameBufferIndex:=iFrameBufferIndex+iLength;
    byteFrameBuffer[iFrameBufferIndex]:=EPICS_ASCII_COMMA; // ,
    iFrameBufferIndex:=iFrameBufferIndex+1;

        IF iFrameBufferIndex>=EPICS_MAX_FRAME_SIZE-25 THEN  //Send before full buffer
            fbTx.AddTail( bPut := ADR(byteFrameBuffer), nWriteCount:=iFrameBufferIndex);(* Put string to the tx fifo *)
            IF NOT fbTx.bOk THEN(* TX fifo overflow => log error *)
             fbLog.Error( sMessage := 'FB_FrameFifo(sender)', nErrID := PLCPRJ_ERROR_SENDFIFO_OVERFLOW );
            END_IF
            iFrameBufferIndex:=0;
        END_IF

    sValue:= LREAL_TO_STRING(pInputDataBuffer^.fDeceleration);
    iLength:=len(str:=sValue);
    memcpy(srcAddr:=ADR(sValue),destAddr:=ADR(byteFrameBuffer[iFrameBufferIndex]),n:=iLength);
    iFrameBufferIndex:=iFrameBufferIndex+iLength;
    byteFrameBuffer[iFrameBufferIndex]:=EPICS_ASCII_COMMA; // ,
    iFrameBufferIndex:=iFrameBufferIndex+1;

        IF iFrameBufferIndex>=EPICS_MAX_FRAME_SIZE-25 THEN  //Send before full buffer
            fbTx.AddTail( bPut := ADR(byteFrameBuffer), nWriteCount:=iFrameBufferIndex);(* Put string to the tx fifo *)
            IF NOT fbTx.bOk THEN(* TX fifo overflow => log error *)
             fbLog.Error( sMessage := 'FB_FrameFifo(sender)', nErrID := PLCPRJ_ERROR_SENDFIFO_OVERFLOW );
            END_IF
            iFrameBufferIndex:=0;
        END_IF

    IF pInputDataBuffer^.bJogFwd THEN
        byteFrameBuffer[iFrameBufferIndex]:=EPICS_ASCII_ONE; // 1
    ELSE
        byteFrameBuffer[iFrameBufferIndex]:=EPICS_ASCII_ZERO; // 0
    END_IF
    iFrameBufferIndex:=iFrameBufferIndex+1;
    byteFrameBuffer[iFrameBufferIndex]:=EPICS_ASCII_COMMA; // ,
    iFrameBufferIndex:=iFrameBufferIndex+1;

        IF iFrameBufferIndex>=EPICS_MAX_FRAME_SIZE-25 THEN  //Send before full buffer
            fbTx.AddTail( bPut := ADR(byteFrameBuffer), nWriteCount:=iFrameBufferIndex);(* Put string to the tx fifo *)
            IF NOT fbTx.bOk THEN(* TX fifo overflow => log error *)
             fbLog.Error( sMessage := 'FB_FrameFifo(sender)', nErrID := PLCPRJ_ERROR_SENDFIFO_OVERFLOW );
            END_IF
            iFrameBufferIndex:=0;
        END_IF

    IF pInputDataBuffer^.bJogBwd THEN
        byteFrameBuffer[iFrameBufferIndex]:=EPICS_ASCII_ONE; // 1
    ELSE
        byteFrameBuffer[iFrameBufferIndex]:=EPICS_ASCII_ZERO; // 0
    END_IF
    iFrameBufferIndex:=iFrameBufferIndex+1;
    byteFrameBuffer[iFrameBufferIndex]:=EPICS_ASCII_COMMA; // ,
    iFrameBufferIndex:=iFrameBufferIndex+1;

        IF iFrameBufferIndex>=EPICS_MAX_FRAME_SIZE-25 THEN  //Send before full buffer
            fbTx.AddTail( bPut := ADR(byteFrameBuffer), nWriteCount:=iFrameBufferIndex);(* Put string to the tx fifo *)
            IF NOT fbTx.bOk THEN(* TX fifo overflow => log error *)
             fbLog.Error( sMessage := 'FB_FrameFifo(sender)', nErrID := PLCPRJ_ERROR_SENDFIFO_OVERFLOW );
            END_IF
            iFrameBufferIndex:=0;
        END_IF

    IF pInputDataBuffer^.bLimitFwd THEN
        byteFrameBuffer[iFrameBufferIndex]:=EPICS_ASCII_ONE; // 1
    ELSE
        byteFrameBuffer[iFrameBufferIndex]:=EPICS_ASCII_ZERO; // 0
    END_IF
    iFrameBufferIndex:=iFrameBufferIndex+1;
    byteFrameBuffer[iFrameBufferIndex]:=EPICS_ASCII_COMMA; // ,
    iFrameBufferIndex:=iFrameBufferIndex+1;

        IF iFrameBufferIndex>=EPICS_MAX_FRAME_SIZE-25 THEN  //Send before full buffer
            fbTx.AddTail( bPut := ADR(byteFrameBuffer), nWriteCount:=iFrameBufferIndex);(* Put string to the tx fifo *)
            IF NOT fbTx.bOk THEN(* TX fifo overflow => log error *)
             fbLog.Error( sMessage := 'FB_FrameFifo(sender)', nErrID := PLCPRJ_ERROR_SENDFIFO_OVERFLOW );
            END_IF
            iFrameBufferIndex:=0;
        END_IF

    IF pInputDataBuffer^.bLimitBwd THEN
        byteFrameBuffer[iFrameBufferIndex]:=EPICS_ASCII_ONE; // 1
    ELSE
        byteFrameBuffer[iFrameBufferIndex]:=EPICS_ASCII_ZERO; // 0
    END_IF
    iFrameBufferIndex:=iFrameBufferIndex+1;
    byteFrameBuffer[iFrameBufferIndex]:=EPICS_ASCII_COMMA; // ,
    iFrameBufferIndex:=iFrameBufferIndex+1;

        IF iFrameBufferIndex>=EPICS_MAX_FRAME_SIZE-25 THEN  //Send before full buffer
            fbTx.AddTail( bPut := ADR(byteFrameBuffer), nWriteCount:=iFrameBufferIndex);(* Put string to the tx fifo *)
            IF NOT fbTx.bOk THEN(* TX fifo overflow => log error *)
             fbLog.Error( sMessage := 'FB_FrameFifo(sender)', nErrID := PLCPRJ_ERROR_SENDFIFO_OVERFLOW );
            END_IF
            iFrameBufferIndex:=0;
        END_IF

    sValue:= LREAL_TO_STRING(pInputDataBuffer^.fOverride);
    iLength:=len(str:=sValue);
    memcpy(srcAddr:=ADR(sValue),destAddr:=ADR(byteFrameBuffer[iFrameBufferIndex]),n:=iLength);
    iFrameBufferIndex:=iFrameBufferIndex+iLength;
    byteFrameBuffer[iFrameBufferIndex]:=EPICS_ASCII_COMMA; // ,
    iFrameBufferIndex:=iFrameBufferIndex+1;

        IF iFrameBufferIndex>=EPICS_MAX_FRAME_SIZE-25 THEN  //Send before full buffer
            fbTx.AddTail( bPut := ADR(byteFrameBuffer), nWriteCount:=iFrameBufferIndex);(* Put string to the tx fifo *)
            IF NOT fbTx.bOk THEN(* TX fifo overflow => log error *)
             fbLog.Error( sMessage := 'FB_FrameFifo(sender)', nErrID := PLCPRJ_ERROR_SENDFIFO_OVERFLOW );
            END_IF
            iFrameBufferIndex:=0;
        END_IF

    IF pInputDataBuffer^.bHomeSensor THEN
        byteFrameBuffer[iFrameBufferIndex]:=EPICS_ASCII_ONE; // 1
    ELSE
        byteFrameBuffer[iFrameBufferIndex]:=EPICS_ASCII_ZERO; // 0
    END_IF
    iFrameBufferIndex:=iFrameBufferIndex+1;
    byteFrameBuffer[iFrameBufferIndex]:=EPICS_ASCII_COMMA; // ,
    iFrameBufferIndex:=iFrameBufferIndex+1;

        IF iFrameBufferIndex>=EPICS_MAX_FRAME_SIZE-25 THEN  //Send before full buffer
            fbTx.AddTail( bPut := ADR(byteFrameBuffer), nWriteCount:=iFrameBufferIndex);(* Put string to the tx fifo *)
            IF NOT fbTx.bOk THEN(* TX fifo overflow => log error *)
             fbLog.Error( sMessage := 'FB_FrameFifo(sender)', nErrID := PLCPRJ_ERROR_SENDFIFO_OVERFLOW );
            END_IF
            iFrameBufferIndex:=0;
        END_IF

    IF pInputDataBuffer^.bEnabled THEN
        byteFrameBuffer[iFrameBufferIndex]:=EPICS_ASCII_ONE; // 1
    ELSE
        byteFrameBuffer[iFrameBufferIndex]:=EPICS_ASCII_ZERO; // 0
    END_IF
    iFrameBufferIndex:=iFrameBufferIndex+1;
    byteFrameBuffer[iFrameBufferIndex]:=EPICS_ASCII_COMMA; // ,
    iFrameBufferIndex:=iFrameBufferIndex+1;

        IF iFrameBufferIndex>=EPICS_MAX_FRAME_SIZE-25 THEN  //Send before full buffer
            fbTx.AddTail( bPut := ADR(byteFrameBuffer), nWriteCount:=iFrameBufferIndex);(* Put string to the tx fifo *)
            IF NOT fbTx.bOk THEN(* TX fifo overflow => log error *)
             fbLog.Error( sMessage := 'FB_FrameFifo(sender)', nErrID := PLCPRJ_ERROR_SENDFIFO_OVERFLOW );
            END_IF
            iFrameBufferIndex:=0;
        END_IF

    IF pInputDataBuffer^.bError THEN
        byteFrameBuffer[iFrameBufferIndex]:=EPICS_ASCII_ONE; // 1
    ELSE
        byteFrameBuffer[iFrameBufferIndex]:=EPICS_ASCII_ZERO; // 0
    END_IF
    iFrameBufferIndex:=iFrameBufferIndex+1;
    byteFrameBuffer[iFrameBufferIndex]:=EPICS_ASCII_COMMA; // ,
    iFrameBufferIndex:=iFrameBufferIndex+1;

        IF iFrameBufferIndex>=EPICS_MAX_FRAME_SIZE-25 THEN  //Send before full buffer
            fbTx.AddTail( bPut := ADR(byteFrameBuffer), nWriteCount:=iFrameBufferIndex);(* Put string to the tx fifo *)
            IF NOT fbTx.bOk THEN(* TX fifo overflow => log error *)
             fbLog.Error( sMessage := 'FB_FrameFifo(sender)', nErrID := PLCPRJ_ERROR_SENDFIFO_OVERFLOW );
            END_IF
            iFrameBufferIndex:=0;
        END_IF

    sValue:= UDINT_TO_STRING(pInputDataBuffer^.nErrorId);
    iLength:=len(str:=sValue);
    memcpy(srcAddr:=ADR(sValue),destAddr:=ADR(byteFrameBuffer[iFrameBufferIndex]),n:=iLength);
    iFrameBufferIndex:=iFrameBufferIndex+iLength;
    byteFrameBuffer[iFrameBufferIndex]:=EPICS_ASCII_COMMA; // ,
    iFrameBufferIndex:=iFrameBufferIndex+1;

        IF iFrameBufferIndex>=EPICS_MAX_FRAME_SIZE-25 THEN  //Send before full buffer
            fbTx.AddTail( bPut := ADR(byteFrameBuffer), nWriteCount:=iFrameBufferIndex);(* Put string to the tx fifo *)
            IF NOT fbTx.bOk THEN(* TX fifo overflow => log error *)
             fbLog.Error( sMessage := 'FB_FrameFifo(sender)', nErrID := PLCPRJ_ERROR_SENDFIFO_OVERFLOW );
            END_IF
            iFrameBufferIndex:=0;
        END_IF

    sValue:= LREAL_TO_STRING(pInputDataBuffer^.fActVelocity);
    iLength:=len(str:=sValue);
    memcpy(srcAddr:=ADR(sValue),destAddr:=ADR(byteFrameBuffer[iFrameBufferIndex]),n:=iLength);
    iFrameBufferIndex:=iFrameBufferIndex+iLength;
    byteFrameBuffer[iFrameBufferIndex]:=EPICS_ASCII_COMMA; // ,
    iFrameBufferIndex:=iFrameBufferIndex+1;

        IF iFrameBufferIndex>=EPICS_MAX_FRAME_SIZE-25 THEN  //Send before full buffer
            fbTx.AddTail( bPut := ADR(byteFrameBuffer), nWriteCount:=iFrameBufferIndex);(* Put string to the tx fifo *)
            IF NOT fbTx.bOk THEN(* TX fifo overflow => log error *)
             fbLog.Error( sMessage := 'FB_FrameFifo(sender)', nErrID := PLCPRJ_ERROR_SENDFIFO_OVERFLOW );
            END_IF
            iFrameBufferIndex:=0;
        END_IF

    sValue:= LREAL_TO_STRING(pInputDataBuffer^.fActPosition);
    iLength:=len(str:=sValue);
    memcpy(srcAddr:=ADR(sValue),destAddr:=ADR(byteFrameBuffer[iFrameBufferIndex]),n:=iLength);
    iFrameBufferIndex:=iFrameBufferIndex+iLength;
    byteFrameBuffer[iFrameBufferIndex]:=EPICS_ASCII_COMMA; // ,
    iFrameBufferIndex:=iFrameBufferIndex+1;

        IF iFrameBufferIndex>=EPICS_MAX_FRAME_SIZE-25 THEN  //Send before full buffer
            fbTx.AddTail( bPut := ADR(byteFrameBuffer), nWriteCount:=iFrameBufferIndex);(* Put string to the tx fifo *)
            IF NOT fbTx.bOk THEN(* TX fifo overflow => log error *)
             fbLog.Error( sMessage := 'FB_FrameFifo(sender)', nErrID := PLCPRJ_ERROR_SENDFIFO_OVERFLOW );
            END_IF
            iFrameBufferIndex:=0;
        END_IF

    sValue:= LREAL_TO_STRING(pInputDataBuffer^.fActDiff);
    iLength:=len(str:=sValue);
    memcpy(srcAddr:=ADR(sValue),destAddr:=ADR(byteFrameBuffer[iFrameBufferIndex]),n:=iLength);
    iFrameBufferIndex:=iFrameBufferIndex+iLength;
    byteFrameBuffer[iFrameBufferIndex]:=EPICS_ASCII_COMMA; // ,
    iFrameBufferIndex:=iFrameBufferIndex+1;

        IF iFrameBufferIndex>=EPICS_MAX_FRAME_SIZE-25 THEN  //Send before full buffer
            fbTx.AddTail( bPut := ADR(byteFrameBuffer), nWriteCount:=iFrameBufferIndex);(* Put string to the tx fifo *)
            IF NOT fbTx.bOk THEN(* TX fifo overflow => log error *)
             fbLog.Error( sMessage := 'FB_FrameFifo(sender)', nErrID := PLCPRJ_ERROR_SENDFIFO_OVERFLOW );
            END_IF
            iFrameBufferIndex:=0;
        END_IF

    IF pInputDataBuffer^.bHomed THEN
        byteFrameBuffer[iFrameBufferIndex]:=EPICS_ASCII_ONE; // 1
    ELSE
        byteFrameBuffer[iFrameBufferIndex]:=EPICS_ASCII_ZERO; // 0
    END_IF
    iFrameBufferIndex:=iFrameBufferIndex+1;
    byteFrameBuffer[iFrameBufferIndex]:=EPICS_ASCII_COMMA; // ,
    iFrameBufferIndex:=iFrameBufferIndex+1;

        IF iFrameBufferIndex>=EPICS_MAX_FRAME_SIZE-25 THEN  //Send before full buffer
            fbTx.AddTail( bPut := ADR(byteFrameBuffer), nWriteCount:=iFrameBufferIndex);(* Put string to the tx fifo *)
            IF NOT fbTx.bOk THEN(* TX fifo overflow => log error *)
             fbLog.Error( sMessage := 'FB_FrameFifo(sender)', nErrID := PLCPRJ_ERROR_SENDFIFO_OVERFLOW );
            END_IF
            iFrameBufferIndex:=0;
        END_IF

    IF pInputDataBuffer^.bBusy THEN
        byteFrameBuffer[iFrameBufferIndex]:=EPICS_ASCII_ONE; // 1
    ELSE
        byteFrameBuffer[iFrameBufferIndex]:=EPICS_ASCII_ZERO; // 0
    END_IF
    iFrameBufferIndex:=iFrameBufferIndex+1;

    bReady:=TRUE;   //Buffer ready for sending!
END_IF

END_FUNCTION_BLOCK

// ---- POUs/FB_StreamBufferToADSBuffer.TcPOU
///#########################################################
///Function Block for parsing of ASCII Stream to binary ADS buffer
/// Library:
///
///
/// Global Variables:
/// - EPICS_MAX_FRAME_SIZE
/// - EPICS_ARRAY_DELIMITER
/// - EPICS_COMMAND_DELIMITER
/// - PLCPRJ_BUFFER_SIZE
///
/// Data types:
///
/// External functions:
///     - TC2_Standard lib
///     - Tc2_Utilities lib
///     - Tc2_System lib
///
///###########################################################
FUNCTION_BLOCK FB_StreamBufferToADSBuffer
VAR
    sVersion: STRING:='0.9.0';
END_VAR
VAR_INPUT
    bExecute: BOOL;
    symbolInfo:SYMINFOSTRUCT;
    nBufferToParseLength:UDINT:=0;
END_VAR
VAR_IN_OUT
    fbLog               : FB_LogFifo;(* Log message fifo *)
    byteASCIIBufferToParse  : ARRAY[0..PLCPRJ_BUFFER_SIZE] OF BYTE;
    byteBinayBufferOutput       : ARRAY[0..PLCPRJ_BUFFER_SIZE] OF BYTE;//Max buffer for input arrays in 'any data type'. Consider max 8 bytes for each char in output string array. Not so nice to hardcode size but to avoid _NEW operator
END_VAR
VAR
    psValue: POINTER TO STRING; //string to point into byte buffer
    nIndex:INT:=0;
    pBuffer:PVOID;
    nInt16Value:INT:=0;
    nUInt16Value:UINT:=0;
    bValue:BOOL:=FALSE;
    r64Value:LREAL:=0.0;
    r32Value:REAL:=0.0;
    nUdInt32Value: UDINT:=0;
    nLInt64Value:LINT:=0;
    stringValue:STRING(255):='';
    sValue:STRING(20):='';
    nByteValue: BYTE:=0;
    nSInt8Value:SINT:=0;
    nDint32Value:DINT:=0;
    nULInt64Value:ULINT:=0;
    sVal: STRING(255);
    nLoopCounter: INT:=0;
    nSize: INT;
    nBufferToParseIndex: INT;
    nAsciiLength: DINT;
    sFind:STRING;
    nIndex2: INT;
    pString: POINTER TO string;
END_VAR

VAR_OUTPUT
    bBusy: BOOL;
    bDone: BOOL;
    bError: BOOL;
    nErrorId: UDINT;
    nBinaryBytesWritten:UDINT:=0;
    nASCIIBytesParsed:UDINT:=0;
END_VAR


bBusy:=TRUE;
bDone:=FALSE;
bError:=FALSE;
IF bExecute THEN
    nBufferToParseIndex:=0;
    nLoopCounter:=0;
    sFind:='                                ';
    memcpy(destAddr:=ADR(sFind),srcAddr:=ADR(byteASCIIBufferToParse[nBufferToParseIndex]),n:=30);    //30 bytes is longer than all current supported data types . NOTE Ascii
    nIndex:=find(STR1:=sFind,STR2:=EPICS_ARRAY_DELIMITER);
    IF nIndex=0 OR nIndex > nBufferToParseLength THEN //Scalar
        nIndex:=find(STR1:=sFind,STR2:=EPICS_COMMAND_DELIMITER);
        IF nIndex>nBufferToParseLength+1 THEN
            nIndex:=UDINT_TO_INT( nBufferToParseLength+1); //Ensure inside buffer
        END_IF
    END_IF

    IF(nBufferToParseLength>0) THEN
        IF NOT (symbolInfo.adsDataType= ADST_STRING OR  symbolInfo.adsDataType=ADST_BIGTYPE OR  symbolInfo.adsDataType=ADST_WSTRING OR symbolInfo.adsDataType=ADST_MAXTYPES OR symbolInfo.adsDataType=ADST_REAL80  OR symbolInfo.adsDataType=ADST_VOID) THEN    //Special cases
            WHILE  nIndex>0 AND symbolInfo.byteSize> nLoopCounter*nSize AND nBufferToParseIndex+nIndex<PLCPRJ_BUFFER_SIZE-255 AND nBufferToParseLength>nBufferToParseIndex DO //-255 to be able to allocate string variable
                sVal:='';
                MEMSET(destAddr:=ADR(sVal),fillByte:=0,n:=20); //No data type will be longer than 20byte
                memcpy(destAddr:=ADR(sVal),srcAddr:=ADR(byteASCIIBufferToParse[nBufferToParseIndex]),n:=nIndex-1);
                sVal[nIndex]:=0;
                CASE symbolInfo.adsDataType OF
                    ADST_INT8: //sint
                        nSize:=1;
                        nSInt8Value:=STRING_TO_SINT(sVal);
                        MEMCPY(destAddr:=ADR(byteBinayBufferOutput[nLoopCounter*nSize]),srcAddr:=ADR(nSInt8Value), nSize);
                    ADST_UINT8:  //byte
                        nSize:=1;
                        nByteValue:=STRING_TO_BYTE(sVal);
                        MEMCPY(destAddr:=ADR(byteBinayBufferOutput[nLoopCounter*nSize]),srcAddr:=ADR(nByteValue), nSize);
                    ADST_INT16:
                        nSize:=2;
                        nInt16Value:=STRING_TO_INT(sVal);
                        MEMCPY(destAddr:=ADR(byteBinayBufferOutput[nLoopCounter*nSize]),srcAddr:=ADR(nInt16Value), nSize);
                    ADST_UINT16:
                        nSize:=2;
                        nUInt16Value:=STRING_TO_UINT(sVal);
                        MEMCPY(destAddr:=ADR(byteBinayBufferOutput[nLoopCounter*nSize]),srcAddr:=ADR(nUInt16Value), nSize);
                    ADST_INT32:  //Dint
                        nSize:=4;
                        nDint32Value:=STRING_TO_DINT(sVal);
                        MEMCPY(destAddr:=ADR(byteBinayBufferOutput[nLoopCounter*nSize]),srcAddr:=ADR(nDint32Value), nSize);
                    ADST_UINT32:
                        nSize:=4;
                        nUdInt32Value:=STRING_TO_UDINT(sVal);
                        MEMCPY(destAddr:=ADR(byteBinayBufferOutput[nLoopCounter*nSize]),srcAddr:=ADR(nUdInt32Value), nSize);
                    ADST_INT64:
                        nSize:=8;
                        nLInt64Value:=STRING_TO_LINT(sVal);
                        MEMCPY(destAddr:=ADR(byteBinayBufferOutput[nLoopCounter*nSize]),srcAddr:=ADR(nLInt64Value), nSize);
                    ADST_UINT64:
                        nSize:=8;
                        nULInt64Value:=STRING_TO_ULINT(sVal);
                        MEMCPY(destAddr:=ADR(byteBinayBufferOutput[nLoopCounter*nSize]),srcAddr:=ADR(nULInt64Value), nSize);
                    ADST_REAL32:
                        nSize:=4;
                        r32Value:=STRING_TO_REAL(sVal);
                        MEMCPY(destAddr:=ADR(byteBinayBufferOutput[nLoopCounter*nSize]),srcAddr:=ADR(r32Value), nSize);
                    ADST_REAL64: //LREAL
                        nSize:=8;
                        r64Value:=STRING_TO_LREAL(sVal);
                        MEMCPY(destAddr:=ADR(byteBinayBufferOutput[nLoopCounter*nSize]),srcAddr:=ADR(r64Value), nSize);
                    ADST_BIT:
                        nSize:=1;
                        IF len(str:=sVal)<4 THEN  //"1" OR "0"
                            bValue:=INT_TO_BOOL(find(str1:=sVal,STR2:='1'));
                        ELSE                        //"TRUE" OR "FALSE"
                            bValue:=STRING_TO_BOOL(sVal);
                        END_IF
                        MEMCPY(destAddr:=ADR(byteBinayBufferOutput[nLoopCounter*nSize]),srcAddr:=ADR(bValue), nSize);   //Must test
                END_CASE
                nBufferToParseIndex:=nBufferToParseIndex+nIndex;
                sFind:='                                ';
                memcpy(destAddr:=ADR(sFind),srcAddr:=ADR(byteASCIIBufferToParse[nBufferToParseIndex]),n:=30);    //30 bytes is longer than all current supported data types ASCII
                nIndex:=find(STR1:=sFind,STR2:=EPICS_ARRAY_DELIMITER);
                IF nIndex=0 THEN
                    nIndex:=find(STR1:=sFind,STR2:=EPICS_COMMAND_DELIMITER);  //Last value in array
                END_IF
                nLoopCounter:=nLoopCounter+1;
            END_WHILE
            nBinaryBytesWritten:=nLoopCounter*nSize;
            nASCIIBytesParsed:= nBufferToParseLength;
        ELSE  //Special cases
            CASE symbolInfo.adsDataType OF
                    ADST_VOID:
                        ; //Data type ADST_VOID not implmented
                    ADST_STRING:
                        IF(symbolInfo.byteSize< PLCPRJ_BUFFER_SIZE) THEN
                            MEMSET(destAddr:=ADR(byteBinayBufferOutput[0]),fillByte:=0,n:=symbolInfo.byteSize);//Clear complete string. Otherwise only a part of the string will be overwritten
                        END_IF
                        MEMCPY(destAddr:=ADR(byteBinayBufferOutput[0]),srcAddr:=ADR(byteASCIIBufferToParse[0]), nBufferToParseLength);
                        nBinaryBytesWritten:=symbolInfo.byteSize; //Allways send complete string
                        nASCIIBytesParsed:= nBufferToParseLength;
                    ADST_WSTRING:
                        ; //Data type ADST_WSTRING not implmented
                    ADST_BIGTYPE:
                        ; //Data type ADST_BIGTYPE not implmented
                    ADST_MAXTYPES:
                        ; //Data type ADST_MAXTYPES not implmented
                    ADST_REAL80:
                        ; //Data type ADST_REAL80 not implmented1
            END_CASE
        END_IF
    END_IF
    bBusy:=FALSE;
    bDone:=TRUE;
ELSE
    bBusy:=FALSE;
    bDone:=FALSE;
    bError:=FALSE;
    nErrorId:=0;
END_IF

END_FUNCTION_BLOCK

// ---- POUs/FB_ValidCommand.TcPOU
FUNCTION_BLOCK FB_ValidCommand
VAR
    sVersion: STRING:='0.9.0';
END_VAR
VAR_INPUT
    pbCommandBuffer : POINTER TO ARRAY[0..PLCPRJ_BUFFER_SIZE] OF BYTE; (* Byte *)
    nBytesInCommandBuffer:UDINT;
END_VAR
VAR_OUTPUT
    bValid:BOOL:=TRUE;
    nIndexEndOfCommand: UDINT;
END_VAR
VAR
    fbFindChar:FB_FindChar;
END_VAR

//Check for end of command (semi colon)
bValid:=FALSE;
fbFindChar(pbBuffer:=pbCommandBuffer,nLength:=nBytesInCommandBuffer,cFind:=EPICS_ASCII_COMMAND_DELIMITER,bDirection:=TRUE);
IF fbFindChar.nIndex>0 AND fbFindChar.nIndex<=nBytesInCommandBuffer THEN
    nIndexEndOfCommand:=fbFindChar.nIndex;
    //Check for read command (?)
    fbFindChar(pbBuffer:=pbCommandBuffer,nLength:=nBytesInCommandBuffer,cFind:=EPICS_ASCII_QUESTIONMARK,bDirection:=TRUE);
    IF fbFindChar.nIndex>0 AND fbFindChar.nIndex<=nBytesInCommandBuffer AND nIndexEndOfCommand>fbFindChar.nIndex THEN //read command
        bValid:=TRUE;
    ELSE
        //Check for write command (=)
        fbFindChar(pbBuffer:=pbCommandBuffer,nLength:=nBytesInCommandBuffer,cFind:=EPICS_ASCII_EQUAL,bDirection:=TRUE);
        IF fbFindChar.nIndex>0 AND fbFindChar.nIndex<=nBytesInCommandBuffer AND nIndexEndOfCommand>fbFindChar.nIndex THEN //write command
            bValid:=TRUE;
        END_IF
    END_IF
END_IF

END_FUNCTION_BLOCK

// ---- POUs/Helper POUs/FB_FindChar.TcPOU
FUNCTION_BLOCK FB_FindChar
VAR
    sVersion: STRING:='0.9.0';
END_VAR
VAR_INPUT
    pbBuffer    : POINTER TO ARRAY[0..PLCPRJ_BUFFER_SIZE] OF BYTE; (* Byte *)
    nLength     : UDINT:=0; // length to search (less than PLCPRJ_BUFFER_SIZE)
    nStartIndex : UDINT:=0;
    cFind       : BYTE; //char to find
    bDirection  : BOOL:=TRUE; // true start from 0, false start from nLength-1
END_VAR
VAR_OUTPUT
    nIndex:UDINT;
END_VAR
VAR
    bFound: BOOL;
END_VAR

nIndex:=-1;
IF nLength>0 AND nStartIndex<nLength AND nStartIndex>=0 THEN
    (*IF bDirection THEN
        nIndex:=0;
    ELSE
        IF nLength<(PLCPRJ_BUFFER_SIZE) THEN
            nIndex:=nLength-1;
        ELSE
            nIndex:=UDINT_TO_INT(PLCPRJ_BUFFER_SIZE-1);
        END_IF
    END_IF*)

    nIndex:=nStartIndex;
    bFound:=FALSE;
    WHILE NOT bFound AND nIndex<nLength AND nIndex<PLCPRJ_BUFFER_SIZE AND nIndex>=0 DO
        IF pbBuffer^[nIndex]= cFind THEN
            bFound:=TRUE;
        ELSE
            IF bDirection THEN
                nIndex:=nIndex+1;
            ELSE
                nIndex:=nIndex-1;
            END_IF
        END_IF
    END_WHILE;
    IF NOT bFound THEN
        nIndex:=-1;
    END_IF
END_IF

END_FUNCTION_BLOCK

// ---- POUs/Static Command support/FB_ParseCommandOption.TcPOU
FUNCTION_BLOCK FB_ParseCommandOption
VAR
    sVersion: STRING:='0.9.0';
END_VAR
VAR_INPUT
    nCommandEndIndex:INT:=0;
END_VAR
VAR
    psCommandBufferString: POINTER TO STRING; //string to point into byte buffer
    nEqualSign: INT;
    nQuestionMark: INT;
END_VAR

VAR_IN_OUT
    byteCommandBuffer   :   ARRAY[0..PLCPRJ_BUFFER_SIZE] OF BYTE;//ADS input buffer
    nBytesInCommandBuffer:DINT:=0;
    nIndexEndOfCommand:DINT:=0;
END_VAR

VAR_OUTPUT
    nErrorId: UDINT;
    bError:BOOL:=FALSE;
    sSubErrorString: STRING;
    sStaticCommand:STRING;
    sStaticValue:STRING;
    bReadCommand:BOOL:=FALSE;
    bWriteCommand:BOOL:=FALSE;
    bWritePersistent:BOOL:=FALSE;
END_VAR

//Parse static command
nErrorId:=0;
bError:=FALSE;
sStaticCommand:='';
sStaticValue:='';
bReadCommand:=FALSE;
bWriteCommand:=FALSE;
bWritePersistent:=FALSE;
psCommandBufferString:=ADR(byteCommandBuffer);

nEqualSign:=find(STR1:=PSTRING_TO_STRING(psCommandBufferString),STR2:=EPICS_WRITE_CMD);
IF nEqualSign>0 AND nEqualSign<nCommandEndIndex THEN
    bWriteCommand:=TRUE;
    //Command
    memcpy(destAddr:=ADR(sStaticCommand[0]),srcAddr:=ADR(byteCommandBuffer[0]),n:=nEqualSign-1);
    memset(destAddr :=ADR(sStaticCommand[nEqualSign-1]),fillByte:=0,n:=1);              //Terminate string
    //Check if persistent
    //IF find(STR1:=sStaticCommand,STR2:=EPICS_STATIC_COMMAND_PERSISTENT)>0 THEN
//      bWritePersistent:=TRUE;
//  END_IF
    //Value
    memcpy(destAddr:=ADR(sStaticValue[0]),srcAddr:=ADR(byteCommandBuffer[nEqualSign]),n:=nCommandEndIndex-nEqualSign-1);
    memset(destAddr :=ADR(sStaticValue[nCommandEndIndex-nEqualSign-1]),fillByte:=0,n:=1); //Terminate string
    IF NOT F_RemoveBytesFromBuffer(nRemoveBytes:= nCommandEndIndex,byteCommandBuffer:=byteCommandBuffer,nBytesInCommandBuffer:=nBytesInCommandBuffer,nIndexEndOfCommand:=nIndexEndOfCommand) THEN
        bError:=TRUE;
        nErrorId:=301;
        sSubErrorString:='State 3: Failed to clear buffer (Parse static command write).';
    END_IF
ELSE
    nQuestionMark:=find(STR1:=PSTRING_TO_STRING(psCommandBufferString),STR2:=EPICS_READ_CMD);
    IF nQuestionMark>0 AND nQuestionMark<nCommandEndIndex THEN
        bReadCommand:=TRUE;
        //Command
        memcpy(destAddr:=ADR(sStaticCommand[0]),srcAddr:=ADR(byteCommandBuffer[0]),n:=nQuestionMark-1);
        memset(destAddr :=ADR(sStaticCommand[nQuestionMark-1]),fillByte:=0,n:=1);               //Terminate string

        //Clean buffer
        IF NOT F_RemoveBytesFromBuffer(nRemoveBytes:= nCommandEndIndex,byteCommandBuffer:=byteCommandBuffer,nBytesInCommandBuffer:=nBytesInCommandBuffer,nIndexEndOfCommand:=nIndexEndOfCommand) THEN
            bError:=TRUE;
            nErrorId:=302;
            sSubErrorString:='State 3: Failed to clear buffer (Parse static command read).';
        END_IF
    END_IF
END_IF

IF NOT (bReadCommand OR  bWriteCommand) THEN
    bError:=TRUE;
    nErrorId:=303;
    sSubErrorString:='State 3: Parsing of static command failed).';
END_IF

END_FUNCTION_BLOCK

// ---- POUs/Helper POUs/F_RemoveBytesFromBuffer.TcPOU
FUNCTION F_RemoveBytesFromBuffer : BOOL
VAR
    sVersion: STRING:='0.9.0';
END_VAR
VAR_INPUT
    nRemoveBytes:UDINT:=0;
END_VAR
VAR_IN_OUT
    byteCommandBuffer   :   ARRAY[0..PLCPRJ_BUFFER_SIZE] OF BYTE;//ADS input buffer
    nBytesInCommandBuffer:DINT:=0;
    nIndexEndOfCommand:DINT:=0;
END_VAR


VAR
    nCommandEndIndex: DINT;
    bRet: BOOL;
END_VAR

//Remove ADS command from buffer
bRet:=FALSE;
IF nRemoveBytes>0 AND (nRemoveBytes< PLCPRJ_BUFFER_SIZE-nRemoveBytes) THEN
    MEMMOVE(srcAddr:=ADR(byteCommandBuffer[nRemoveBytes]),destAddr:=ADR(byteCommandBuffer[0]),n:= nBytesInCommandBuffer-nRemoveBytes); //remove ADSPORT command from buffer
    MEMSET(destAddr:=ADR(byteCommandBuffer[nBytesInCommandBuffer-nRemoveBytes]),fillByte:=0,n:=nRemoveBytes); //reset buffer
    nBytesInCommandBuffer:=nBytesInCommandBuffer-nRemoveBytes;
    nIndexEndOfCommand:=nIndexEndOfCommand-nRemoveBytes;
    bRet:=TRUE;
END_IF
F_RemoveBytesFromBuffer:=bREt;
RETURN;

END_FUNCTION

// ---- POUs/Static Command support/FB_ParseStringToSymInfo.TcPOU
FUNCTION_BLOCK FB_ParseStringToSymInfo
VAR
    sVersion: STRING:='0.9.0';
END_VAR
VAR_INPUT
    sAdress:STRING:='';
END_VAR
VAR
    sTemp: STRING;
    nEqualSign: INT;
    nComma:INT:=0;
    stemp1: STRING(255);
    sTemp2: STRING(255);
    sTemp3: STRING(255);
    sTemp4: STRING(255);
    sVal:STRING;
    nQuestionSign: INT;
END_VAR

VAR_OUTPUT
    nErrorId: UDINT;
    bError:BOOL:=FALSE;
    sSubErrorString: STRING;
    stSymInfo:SYMINFOSTRUCT;
END_VAR

//Should look like "ADR=idxgrp,idxoff,size,type/"   => ADR=1,2,3,4/
(*
Type:
ADST_BIT             = 33 (&H21)
ADST_INT8            = 16 (&H10)
ADST_INT16           = 2
ADST_INT32           = 3
ADST_INT64           = 20 (&H14)
ADST_UINT8           = 17 (&H11)
ADST_UINT16          = 18 (&H12)
ADST_UINT32          = 19 (&H13)
ADST_UINT64          = 21 (&H15)
ADST_REAL32          = 4
ADST_REAL64          = 5
ADST_REAL80          = 32 (&H20)
ADST_BIGTYPE         = 65 (&H41)
ADST_VOID            = 0
*)

//parse , delimited file to syminfo struct
    bError:=TRUE;
    nErrorId:=401;
    sSubErrorString:='Parsing of absolute adress failed';
    stSymInfo.adsDataType:=0;
    stSymInfo.byteSize:=0;
    stSymInfo.idxGroup:=0;
    stSymInfo.idxOffset:=0;
    nComma:=find(STR1:=sAdress,STR2:=EPICS_ARRAY_DELIMITER);
    IF  nComma>0 THEN
        sVal:=left(STR:=sAdress,size:=nComma);
        stSymInfo.idxGroup:=STRING_TO_UDINT(sVal);
        sTemp1:=right(STR:=sAdress,size:=len(sAdress)-nComma);
        //nRemove:=nRemove+nComma+1;
        nComma:=find(STR1:=sTemp1,STR2:=EPICS_ARRAY_DELIMITER);
        IF  nComma>0 THEN
            sVal:=left(STR:=sTemp1,size:=nComma);
            stSymInfo.idxOffset:=STRING_TO_UDINT(sVal);
            sTemp2:=right(STR:=sTemp1,size:=len(sTemp1)-nComma);
            //nRemove:=nRemove+nComma+1;
            nComma:=find(STR1:=sTemp2,STR2:=EPICS_ARRAY_DELIMITER); //last
            IF  nComma>0 THEN
                sVal:=left(STR:=sTemp2,size:=nComma);
                stSymInfo.byteSize:=STRING_TO_UDINT(sVal);
                sTemp3:=right(STR:=sTemp2,size:=len(sTemp2)-nComma);
                //nRemove:=nRemove+nComma+1;
                nComma:=len(sTemp3);
                IF nComma>0 THEN
                    stSymInfo.adsDataType:=STRING_TO_INT(sTemp3);
                    //nRemove:=nRemove+nComma+1;
                    bError:=FALSE;
                    sSubErrorString:='';
                    nErrorId:=0;
                END_IF
            END_IF
        END_IF
    END_IF

END_FUNCTION_BLOCK

// ---- POUs/FB_ServerConnection.TcPOU
///#########################################################
/// FB that handles one TCP/IP client connection. The code is based on Beckhoff sample code and only minor changes have been made for the EPICS interface.
///
///
/// Library:
///
///
/// Global Variables:
/// - EPICS_MAX_FRAME_SIZE
/// - EPICS_ARRAY_DELIMITER
/// - EPICS_COMMAND_DELIMITER
/// - PLCPRJ_BUFFER_SIZE
///
/// Data types:
///
/// External functions:
///     - TC2_Standard lib
///     - Tc2_Utilities lib
///     - Tc2_System lib
///
///
///###########################################################
FUNCTION_BLOCK FB_ServerConnection
VAR
    sVersion: STRING:='0.9.1';
END_VAR
VAR_IN_OUT
    fbTx            : FB_FrameFifo;(* TX fifo *)
    fbRx            : FB_FrameFifo;(* RX fifo *)
    fbLog           : FB_LogFifo;(* Log message fifo *)
    hListener       : T_HSOCKET;(* Listener socket handle *)
    bReset          : BOOL;
END_VAR
VAR_INPUT
    sSrvNetID       : T_AmsNetID    := '';(* TwinCAT TCP/IP server network address *)
    bEnable         : BOOL          := FALSE;(* TRUE => connect and exchange data, FALSE => disconnect *)
    tReconnect      : TIME          := T#1S;(* Accept new connection (reconnect) after this time *)
    bLog            : BOOL          := FALSE;(* TRUE => Enable log message output, FALSE => Disable *)
    sPrefix         : STRING        := 'SERVERx::';(* Log message description string (allows the identification of log message source) *)
END_VAR
VAR_OUTPUT
    bAccepted       : BOOL          := FALSE;(* Accepted connection status *)
END_VAR
VAR
    fbAccept        : FB_SocketAccept;
    fbClose         : FB_SocketClose;
    fbReceive       : FB_SocketReceive;
    fbSend          : FB_SocketSend;
    eStep           : E_ConnectionSteps;
    bSndBusy        : BOOL;(* Tx state *)
    bRcvBusy        : BOOL;(* Rx state *)
    bDisconnect     : BOOL;(* Disconnect flag, if set the socket will be closed *)

    fbAcceptTimer   : TON;(* Accept poll timer *)
    fbPollTimer     : TON;(* Receive poll timer *)
    fbRequestTimer  : TON;(* Request timeout timer *)

    rxBuffer        : ARRAY[0..PLCPRJ_BUFFER_SIZE] OF BYTE;
    bTxFrame        : ARRAY[0..EPICS_MAX_FRAME_SIZE+5] OF BYTE;
    sTxBuffer       : POINTER TO STRING; //TEMP
    nTxFrameReadLength  : UDINT;
    bRxFrame        : ARRAY[0..PLCPRJ_BUFFER_SIZE] OF BYTE;
    cbReceived      : UDINT;
    nLenOfString    : UDINT;(* String length inclusive the null delimiter *)
    bEndOfString    : BOOL := FALSE;
    bGetMoreData: BOOL;
    nTotalTxFrameReadLength: DINT;
END_VAR


CASE eStep OF
    eCONNECTION_STATE_IDLE:
        IF bEnable XOR bAccepted THEN
            IF bEnable THEN
                fbAcceptTimer( IN := TRUE );
                IF fbAcceptTimer.Q THEN

                    fbTx.Clear( sPrefix := CONCAT( sPrefix, 'FB_FrameFifo(sender)::' ), bLog := bLog );(* Clear send fifo *)
                    fbRx.Clear( sPrefix := CONCAT( sPrefix, 'FB_FrameFifo(receiver)::' ), bLog := bLog );(* Clear receiver fifo *)
                    fbLog.Clear( sPrefix := sPrefix, bLog := bLog );(* Clear log fifo *)
                    bSndBusy := FALSE;
                    bRcvBusy := FALSE;
                    bDisconnect := FALSE;
                    cbReceived := 0;

                    fbPollTimer( IN := FALSE, PT := T#0S );
                    fbRequestTimer( IN := FALSE, PT := PLCPRJ_RECEIVE_TIMEOUT );
                    fbAcceptTimer( IN := FALSE, PT := tReconnect );


